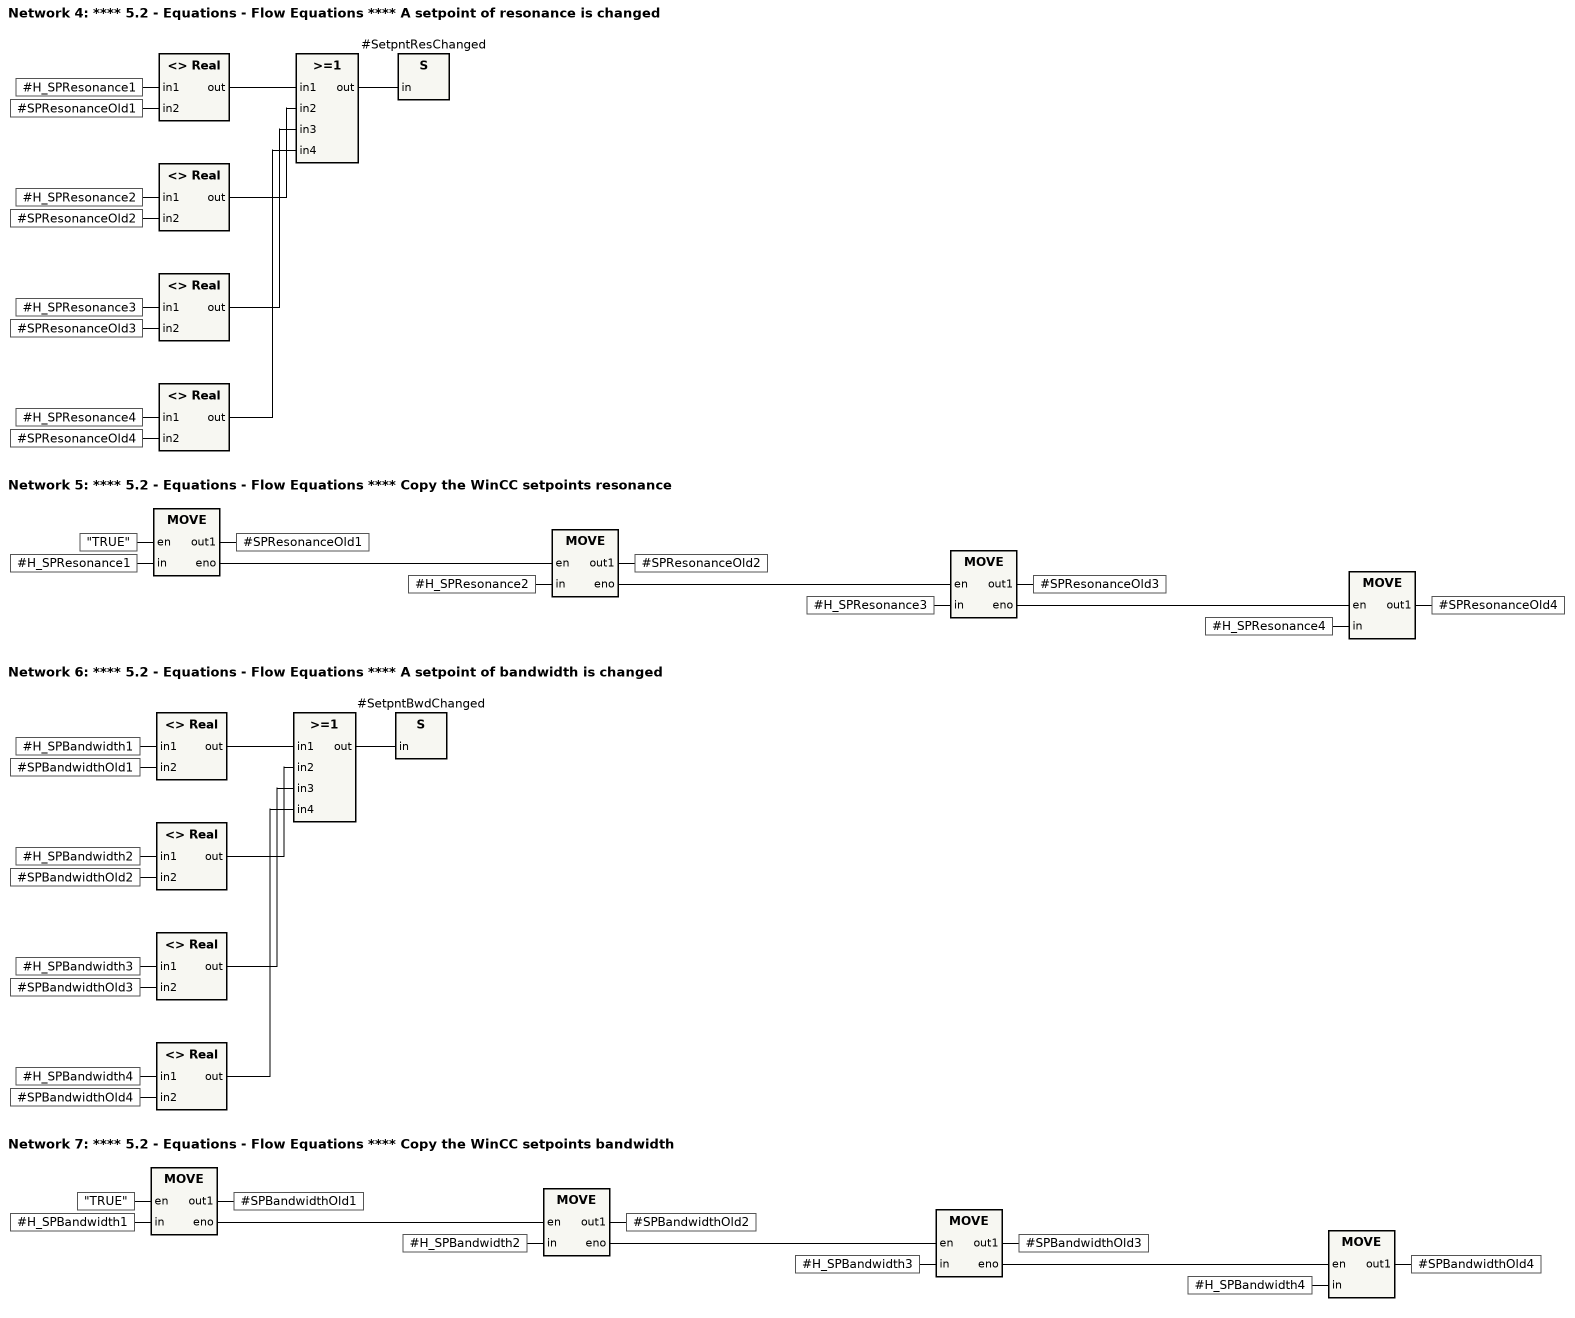
   IF (#H_SPResonance1 <> #SPResonanceOld1) OR (#H_SPResonance2 <> #SPResonanceOld2) OR (#H_SPResonance3 <> #SPResonanceOld3) OR (#H_SPResonance4 <> #SPResonanceOld4) THEN
       #SetpntResChanged := TRUE;
   END_IF;
END_REGION

REGION Network 5: **** 5.2 - Equations - Flow Equations **** Copy the WinCC setpoints resonance
   // Copy the WinCC setpoints resonance
   // ENO of a box is taken as its EN; it also drops when the box reports an error
   IF "TRUE" THEN
       #SPResonanceOld1 := #H_SPResonance1;
       #SPResonanceOld2 := #H_SPResonance2;
       #SPResonanceOld3 := #H_SPResonance3;
       #SPResonanceOld4 := #H_SPResonance4;
   END_IF;
END_REGION

REGION Network 6: **** 5.2 - Equations - Flow Equations **** A setpoint of bandwidth is changed
   // A setpoint of bandwidth is changed
   IF (#H_SPBandwidth1 <> #SPBandwidthOld1) OR (#H_SPBandwidth2 <> #SPBandwidthOld2) OR (#H_SPBandwidth3 <> #SPBandwidthOld3) OR (#H_SPBandwidth4 <> #SPBandwidthOld4) THEN
       #SetpntBwdChanged := TRUE;
   END_IF;
END_REGION

REGION Network 7: **** 5.2 - Equations - Flow Equations **** Copy the WinCC setpoints bandwidth
   // Copy the WinCC setpoints bandwidth
   // ENO of a box is taken as its EN; it also drops when the box reports an error
   IF "TRUE" THEN
       #SPBandwidthOld1 := #H_SPBandwidth1;
       #SPBandwidthOld2 := #H_SPBandwidth2;
       #SPBandwidthOld3 := #H_SPBandwidth3;
       #SPBandwidthOld4 := #H_SPBandwidth4;
   END_IF;
END_REGION

REGION Network 8: **** 5.2 - Equations - Flow Equations **** Selection Set-point 1
   // Selection Set-point 1
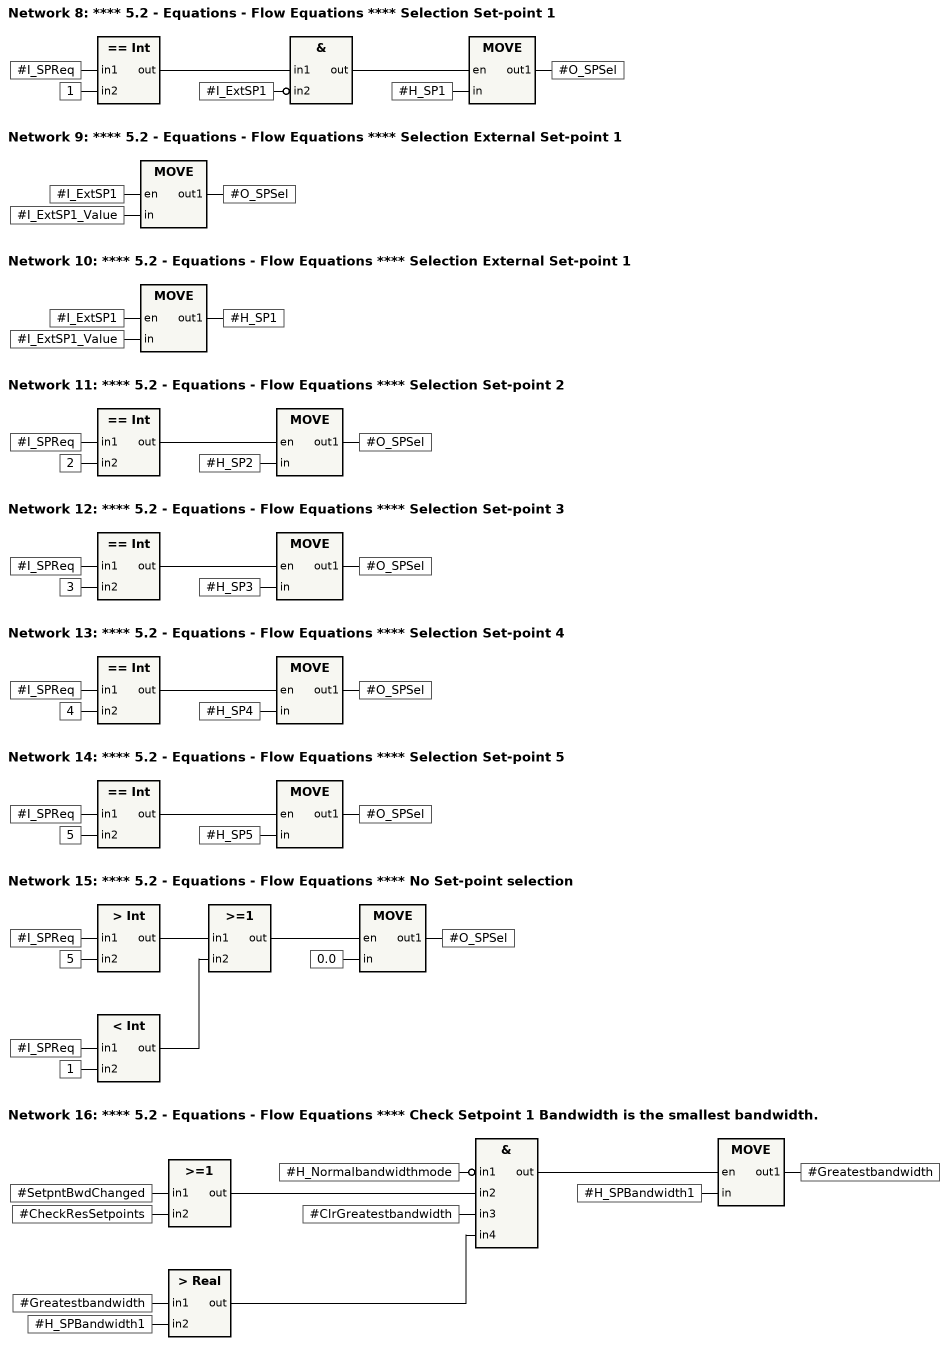
   IF (#I_SPReq = 1) AND NOT #I_ExtSP1 THEN #O_SPSel := #H_SP1; END_IF;
END_REGION

REGION Network 9: **** 5.2 - Equations - Flow Equations **** Selection External Set-point 1
   // Selection External Set-point 1
   IF #I_ExtSP1 THEN #O_SPSel := #I_ExtSP1_Value; END_IF;
END_REGION

REGION Network 10: **** 5.2 - Equations - Flow Equations **** Selection External Set-point 1
   // Selection External Set-point 1
   IF #I_ExtSP1 THEN #H_SP1 := #I_ExtSP1_Value; END_IF;
END_REGION

REGION Network 11: **** 5.2 - Equations - Flow Equations **** Selection Set-point 2
   // Selection Set-point 2
   IF #I_SPReq = 2 THEN #O_SPSel := #H_SP2; END_IF;
END_REGION

REGION Network 12: **** 5.2 - Equations - Flow Equations **** Selection Set-point 3
   // Selection Set-point 3
   IF #I_SPReq = 3 THEN #O_SPSel := #H_SP3; END_IF;
END_REGION

REGION Network 13: **** 5.2 - Equations - Flow Equations **** Selection Set-point 4
   // Selection Set-point 4
   IF #I_SPReq = 4 THEN #O_SPSel := #H_SP4; END_IF;
END_REGION

REGION Network 14: **** 5.2 - Equations - Flow Equations **** Selection Set-point 5
   // Selection Set-point 5
   IF #I_SPReq = 5 THEN #O_SPSel := #H_SP5; END_IF;
END_REGION

REGION Network 15: **** 5.2 - Equations - Flow Equations **** No Set-point selection
   // No Set-point selection
   IF (#I_SPReq > 5) OR (#I_SPReq < 1) THEN #O_SPSel := 0.0; END_IF;
END_REGION

REGION Network 16: **** 5.2 - Equations - Flow Equations **** Check Setpoint 1 Bandwidth is the smallest bandwidth.
   // Check Setpoint 1 Bandwidth is the smallest bandwidth.
   IF NOT #H_Normalbandwidthmode AND (#SetpntBwdChanged OR #CheckResSetpoints) AND #ClrGreatestbandwidth AND (#Greatestbandwidth > #H_SPBandwidth1) THEN
       #Greatestbandwidth := #H_SPBandwidth1;
   END_IF;
END_REGION

REGION Network 17: **** 5.2 - Equations - Flow Equations **** Check Setpoint 2 Bandwidth is the smallest bandwidth.
   // Check Setpoint 2 Bandwidth is the smallest bandwidth.
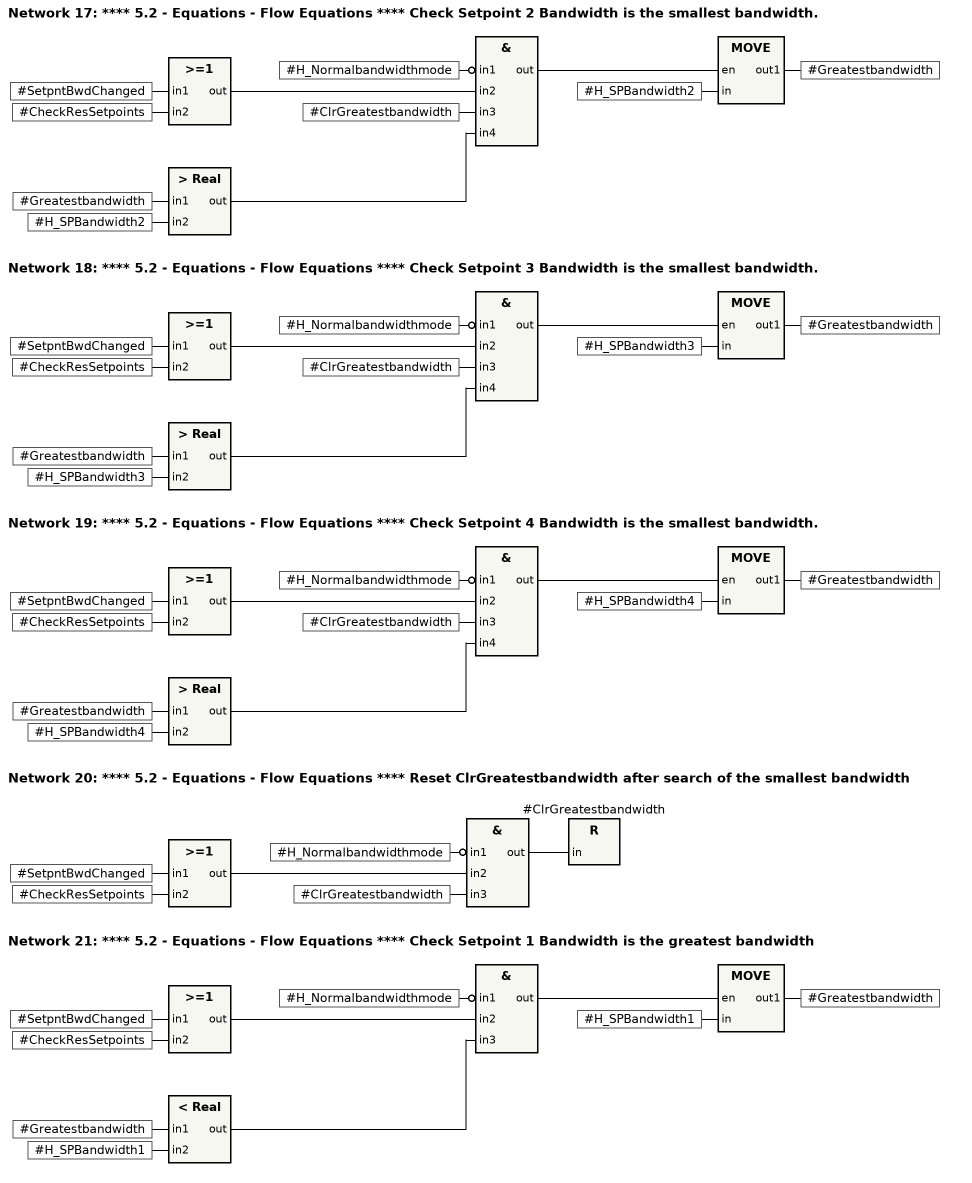
   IF NOT #H_Normalbandwidthmode AND (#SetpntBwdChanged OR #CheckResSetpoints) AND #ClrGreatestbandwidth AND (#Greatestbandwidth > #H_SPBandwidth2) THEN
       #Greatestbandwidth := #H_SPBandwidth2;
   END_IF;
END_REGION

REGION Network 18: **** 5.2 - Equations - Flow Equations **** Check Setpoint 3 Bandwidth is the smallest bandwidth.
   // Check Setpoint 3 Bandwidth is the smallest bandwidth.
   IF NOT #H_Normalbandwidthmode AND (#SetpntBwdChanged OR #CheckResSetpoints) AND #ClrGreatestbandwidth AND (#Greatestbandwidth > #H_SPBandwidth3) THEN
       #Greatestbandwidth := #H_SPBandwidth3;
   END_IF;
END_REGION

REGION Network 19: **** 5.2 - Equations - Flow Equations **** Check Setpoint 4 Bandwidth is the smallest bandwidth.
   // Check Setpoint 4 Bandwidth is the smallest bandwidth.
   IF NOT #H_Normalbandwidthmode AND (#SetpntBwdChanged OR #CheckResSetpoints) AND #ClrGreatestbandwidth AND (#Greatestbandwidth > #H_SPBandwidth4) THEN
       #Greatestbandwidth := #H_SPBandwidth4;
   END_IF;
END_REGION

REGION Network 20: **** 5.2 - Equations - Flow Equations **** Reset ClrGreatestbandwidth after search of the smallest bandwidth
   // Reset ClrGreatestbandwidth after search of the smallest bandwidth
   IF NOT #H_Normalbandwidthmode AND (#SetpntBwdChanged OR #CheckResSetpoints) AND #ClrGreatestbandwidth THEN
       #ClrGreatestbandwidth := FALSE;
   END_IF;
END_REGION

REGION Network 21: **** 5.2 - Equations - Flow Equations **** Check Setpoint 1 Bandwidth is the greatest bandwidth
   // Check Setpoint 1 Bandwidth is the greatest bandwidth
   IF NOT #H_Normalbandwidthmode AND (#SetpntBwdChanged OR #CheckResSetpoints) AND (#Greatestbandwidth < #H_SPBandwidth1) THEN
       #Greatestbandwidth := #H_SPBandwidth1;
   END_IF;
END_REGION

REGION Network 22: **** 5.2 - Equations - Flow Equations **** Check Setpoint 2 Bandwidth is the greatest bandwidth
   // Check Setpoint 2 Bandwidth is the greatest bandwidth
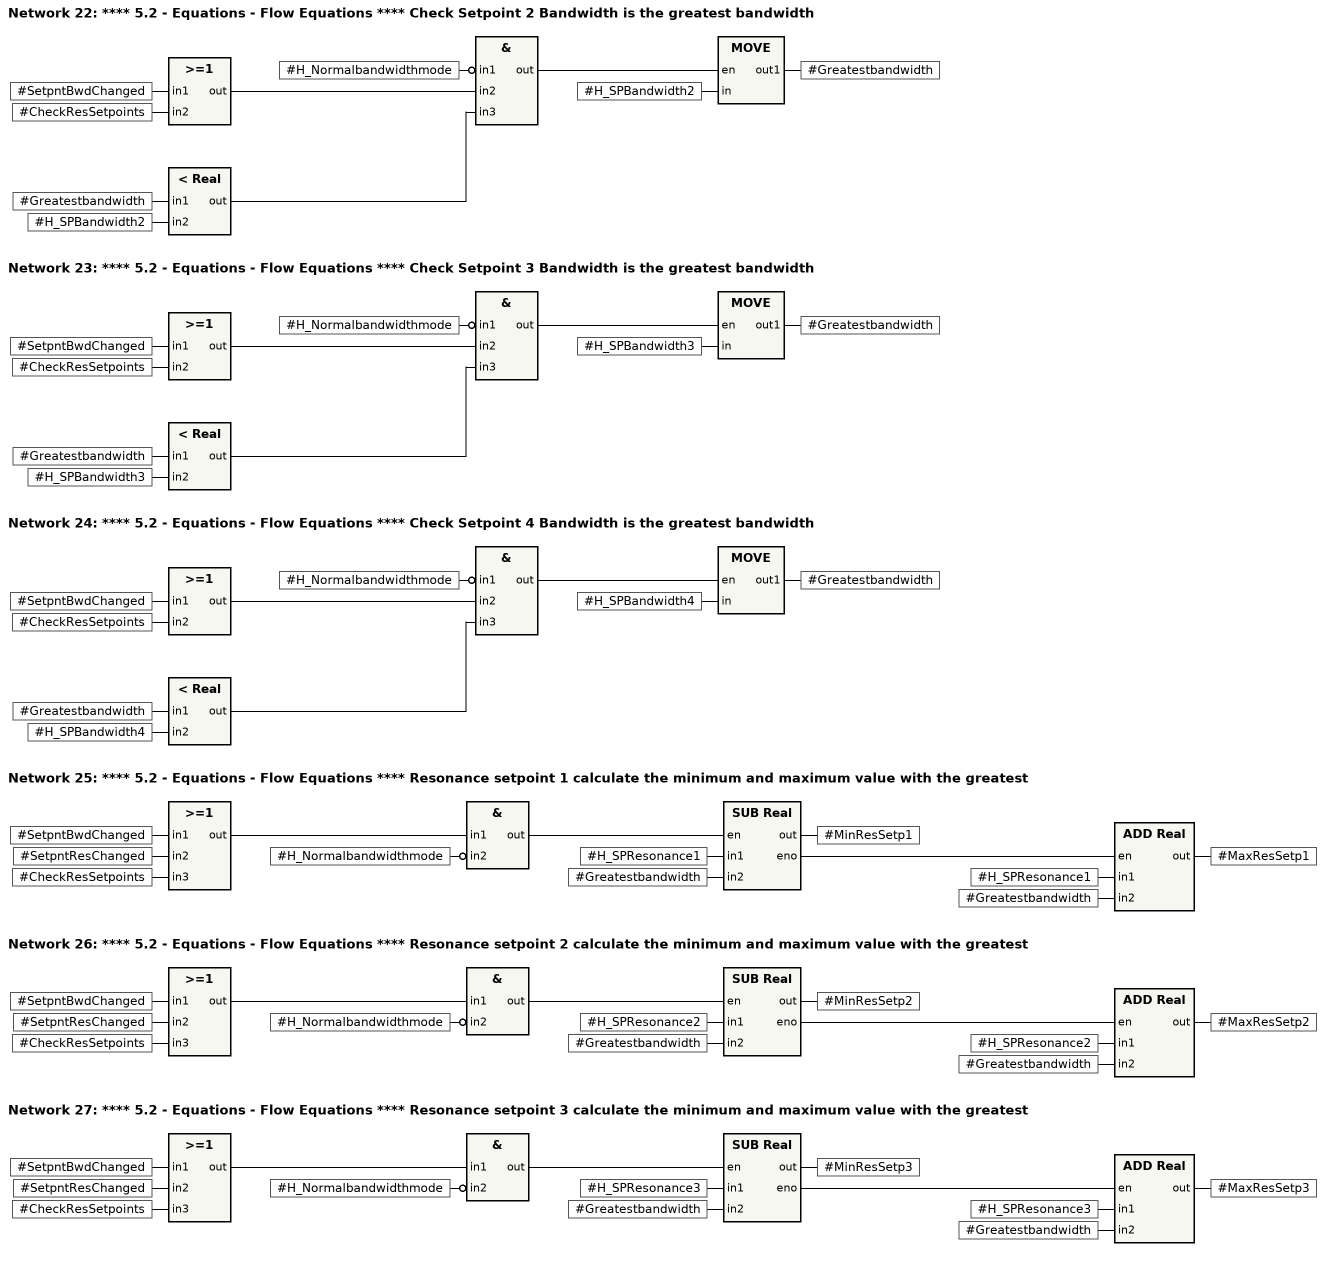
   IF NOT #H_Normalbandwidthmode AND (#SetpntBwdChanged OR #CheckResSetpoints) AND (#Greatestbandwidth < #H_SPBandwidth2) THEN
       #Greatestbandwidth := #H_SPBandwidth2;
   END_IF;
END_REGION

REGION Network 23: **** 5.2 - Equations - Flow Equations **** Check Setpoint 3 Bandwidth is the greatest bandwidth
   // Check Setpoint 3 Bandwidth is the greatest bandwidth
   IF NOT #H_Normalbandwidthmode AND (#SetpntBwdChanged OR #CheckResSetpoints) AND (#Greatestbandwidth < #H_SPBandwidth3) THEN
       #Greatestbandwidth := #H_SPBandwidth3;
   END_IF;
END_REGION

REGION Network 24: **** 5.2 - Equations - Flow Equations **** Check Setpoint 4 Bandwidth is the greatest bandwidth
   // Check Setpoint 4 Bandwidth is the greatest bandwidth
   IF NOT #H_Normalbandwidthmode AND (#SetpntBwdChanged OR #CheckResSetpoints) AND (#Greatestbandwidth < #H_SPBandwidth4) THEN
       #Greatestbandwidth := #H_SPBandwidth4;
   END_IF;
END_REGION

REGION Network 25: **** 5.2 - Equations - Flow Equations **** Resonance setpoint 1 calculate the minimum and maximum value with the greatest
   // Resonance setpoint 1 calculate the minimum and maximum value with the greatest 
   // bandwidth
   // ENO of a box is taken as its EN; it also drops when the box reports an error
   IF (#SetpntBwdChanged OR #SetpntResChanged OR #CheckResSetpoints) AND NOT #H_Normalbandwidthmode THEN
       #MinResSetp1 := #H_SPResonance1 - #Greatestbandwidth;
       #MaxResSetp1 := #H_SPResonance1 + #Greatestbandwidth;
   END_IF;
END_REGION

REGION Network 26: **** 5.2 - Equations - Flow Equations **** Resonance setpoint 2 calculate the minimum and maximum value with the greatest
   // Resonance setpoint 2 calculate the minimum and maximum value with the greatest 
   // bandwidth
   // ENO of a box is taken as its EN; it also drops when the box reports an error
   IF (#SetpntBwdChanged OR #SetpntResChanged OR #CheckResSetpoints) AND NOT #H_Normalbandwidthmode THEN
       #MinResSetp2 := #H_SPResonance2 - #Greatestbandwidth;
       #MaxResSetp2 := #H_SPResonance2 + #Greatestbandwidth;
   END_IF;
END_REGION

REGION Network 27: **** 5.2 - Equations - Flow Equations **** Resonance setpoint 3 calculate the minimum and maximum value with the greatest
   // Resonance setpoint 3 calculate the minimum and maximum value with the greatest 
   // bandwidth
   // ENO of a box is taken as its EN; it also drops when the box reports an error
   IF (#SetpntBwdChanged OR #SetpntResChanged OR #CheckResSetpoints) AND NOT #H_Normalbandwidthmode THEN
       #MinResSetp3 := #H_SPResonance3 - #Greatestbandwidth;
       #MaxResSetp3 := #H_SPResonance3 + #Greatestbandwidth;
   END_IF;
END_REGION

REGION Network 28: **** 5.2 - Equations - Flow Equations **** Resonance setpoint 4 calculate the minimum and maximum value with the greatest
   // Resonance setpoint 4 calculate the minimum and maximum value with the greatest 
   // bandwidth
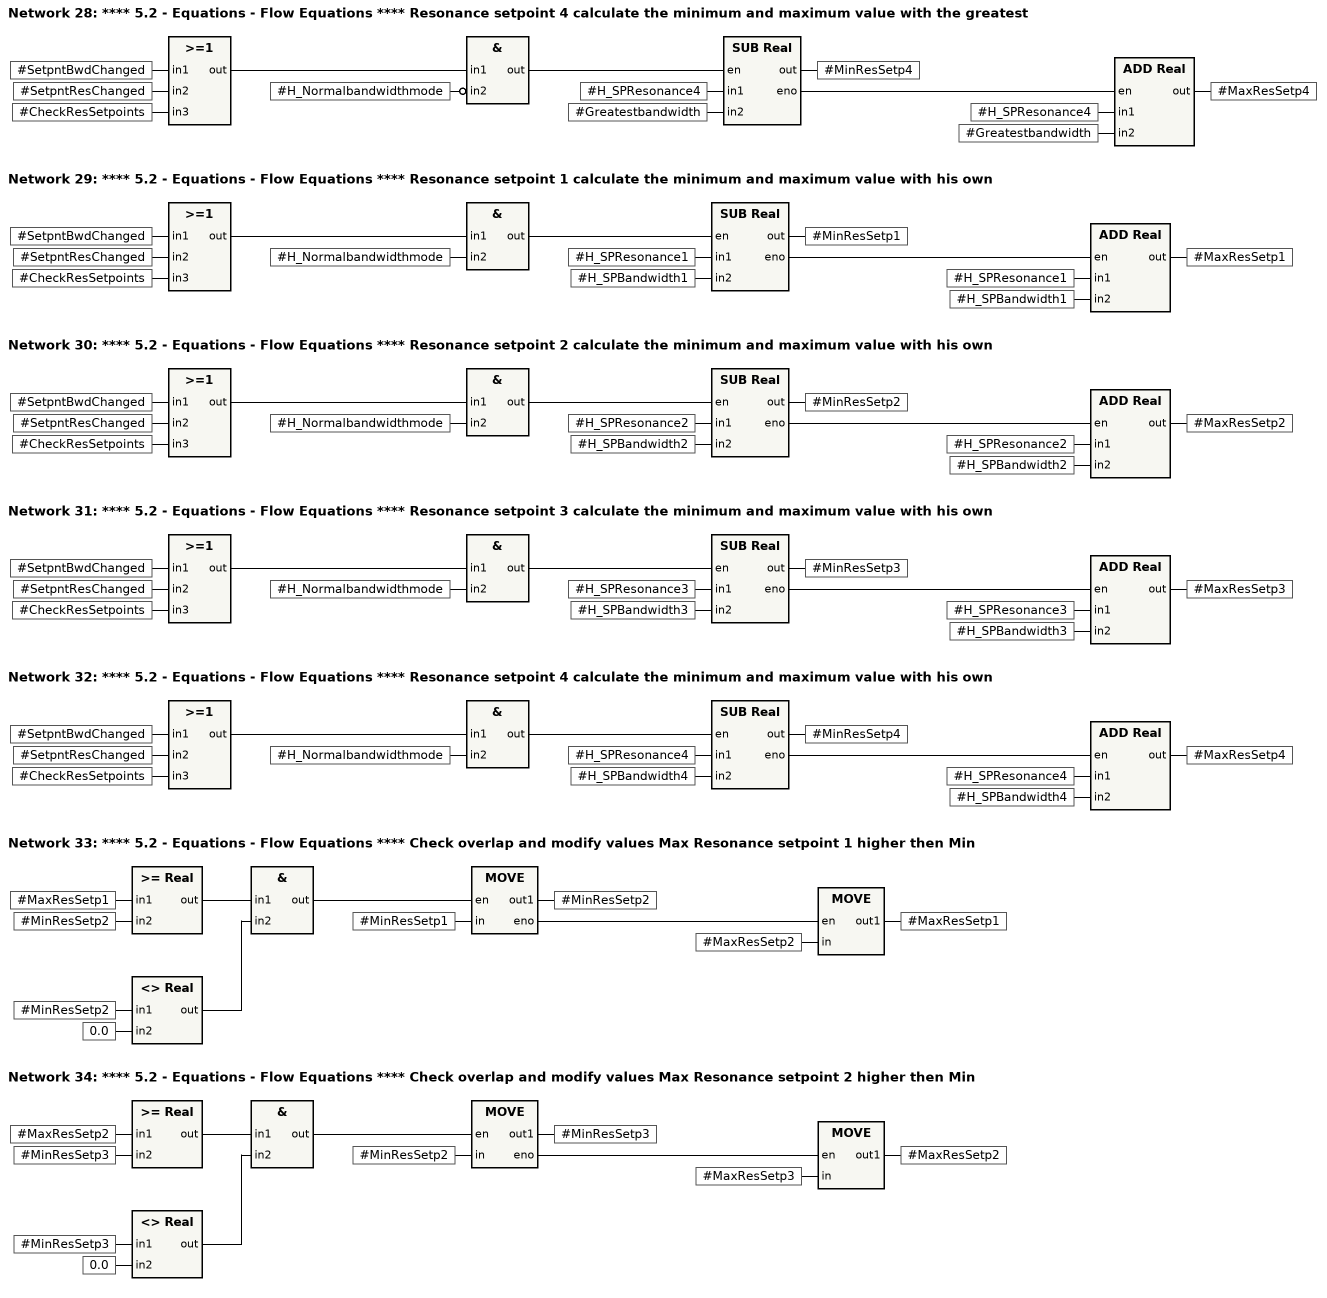
   // ENO of a box is taken as its EN; it also drops when the box reports an error
   IF (#SetpntBwdChanged OR #SetpntResChanged OR #CheckResSetpoints) AND NOT #H_Normalbandwidthmode THEN
       #MinResSetp4 := #H_SPResonance4 - #Greatestbandwidth;
       #MaxResSetp4 := #H_SPResonance4 + #Greatestbandwidth;
   END_IF;
END_REGION

REGION Network 29: **** 5.2 - Equations - Flow Equations **** Resonance setpoint 1 calculate the minimum and maximum value with his own
   // Resonance setpoint 1 calculate the minimum and maximum value with his own 
   // bandwidth
   // ENO of a box is taken as its EN; it also drops when the box reports an error
   IF (#SetpntBwdChanged OR #SetpntResChanged OR #CheckResSetpoints) AND #H_Normalbandwidthmode THEN
       #MinResSetp1 := #H_SPResonance1 - #H_SPBandwidth1;
       #MaxResSetp1 := #H_SPResonance1 + #H_SPBandwidth1;
   END_IF;
END_REGION

REGION Network 30: **** 5.2 - Equations - Flow Equations **** Resonance setpoint 2 calculate the minimum and maximum value with his own
   // Resonance setpoint 2 calculate the minimum and maximum value with his own 
   // bandwidth
   // ENO of a box is taken as its EN; it also drops when the box reports an error
   IF (#SetpntBwdChanged OR #SetpntResChanged OR #CheckResSetpoints) AND #H_Normalbandwidthmode THEN
       #MinResSetp2 := #H_SPResonance2 - #H_SPBandwidth2;
       #MaxResSetp2 := #H_SPResonance2 + #H_SPBandwidth2;
   END_IF;
END_REGION

REGION Network 31: **** 5.2 - Equations - Flow Equations **** Resonance setpoint 3 calculate the minimum and maximum value with his own
   // Resonance setpoint 3 calculate the minimum and maximum value with his own 
   // bandwidth
   // ENO of a box is taken as its EN; it also drops when the box reports an error
   IF (#SetpntBwdChanged OR #SetpntResChanged OR #CheckResSetpoints) AND #H_Normalbandwidthmode THEN
       #MinResSetp3 := #H_SPResonance3 - #H_SPBandwidth3;
       #MaxResSetp3 := #H_SPResonance3 + #H_SPBandwidth3;
   END_IF;
END_REGION

REGION Network 32: **** 5.2 - Equations - Flow Equations **** Resonance setpoint 4 calculate the minimum and maximum value with his own
   // Resonance setpoint 4 calculate the minimum and maximum value with his own 
   // bandwidth
   // ENO of a box is taken as its EN; it also drops when the box reports an error
   IF (#SetpntBwdChanged OR #SetpntResChanged OR #CheckResSetpoints) AND #H_Normalbandwidthmode THEN
       #MinResSetp4 := #H_SPResonance4 - #H_SPBandwidth4;
       #MaxResSetp4 := #H_SPResonance4 + #H_SPBandwidth4;
   END_IF;
END_REGION

REGION Network 33: **** 5.2 - Equations - Flow Equations **** Check overlap and modify values Max Resonance setpoint 1 higher then Min
   // Check overlap and modify values Max Resonance setpoint 1 higher then Min 
   // Resonance setpoint 2
   // ENO of a box is taken as its EN; it also drops when the box reports an error
   #_w1 := (#MaxResSetp1 >= #MinResSetp2) AND (#MinResSetp2 <> 0.0);
   IF #_w1 THEN
       #MinResSetp2 := #MinResSetp1;
       #MaxResSetp1 := #MaxResSetp2;
   END_IF;
END_REGION

REGION Network 34: **** 5.2 - Equations - Flow Equations **** Check overlap and modify values Max Resonance setpoint 2 higher then Min
   // Check overlap and modify values Max Resonance setpoint 2 higher then Min 
   // Resonance setpoint 3
   // ENO of a box is taken as its EN; it also drops when the box reports an error
   #_w1 := (#MaxResSetp2 >= #MinResSetp3) AND (#MinResSetp3 <> 0.0);
   IF #_w1 THEN
       #MinResSetp3 := #MinResSetp2;
       #MaxResSetp2 := #MaxResSetp3;
   END_IF;
END_REGION

REGION Network 35: **** 5.2 - Equations - Flow Equations **** Check overlap and modify values Max Resonance setpoint 3 higher then Min
   // Check overlap and modify values Max Resonance setpoint 3 higher then Min 
   // Resonance setpoint 4
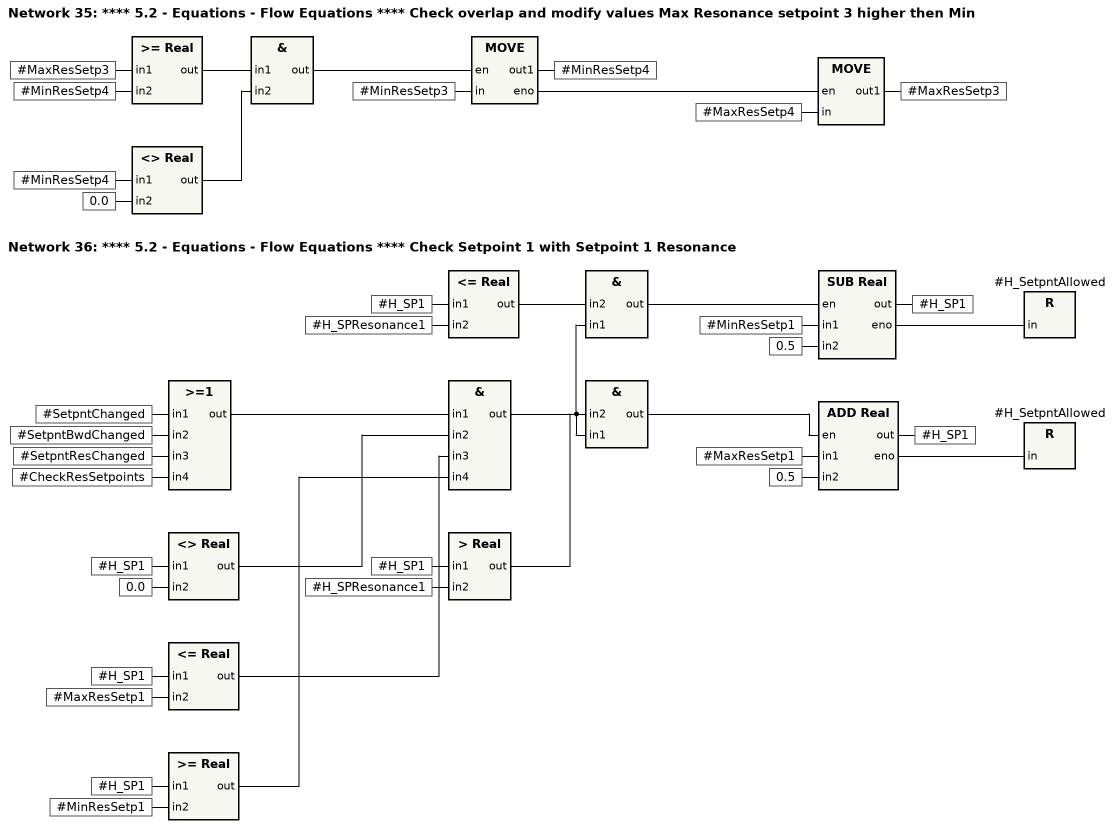
   // ENO of a box is taken as its EN; it also drops when the box reports an error
   #_w1 := (#MaxResSetp3 >= #MinResSetp4) AND (#MinResSetp4 <> 0.0);
   IF #_w1 THEN
       #MinResSetp4 := #MinResSetp3;
       #MaxResSetp3 := #MaxResSetp4;
   END_IF;
END_REGION

REGION Network 36: **** 5.2 - Equations - Flow Equations **** Check Setpoint 1 with Setpoint 1 Resonance
   // Check Setpoint 1 with Setpoint 1 Resonance 
   // Setpoint 1 is no longer allowed, calculate prefered allowed setpoint 1
   // ENO of a box is taken as its EN; it also drops when the box reports an error
   #_w1 := (#SetpntChanged OR #SetpntBwdChanged OR #SetpntResChanged OR #CheckResSetpoints) AND (#H_SP1 <> 0.0) AND (#H_SP1 <= #MaxResSetp1) AND (#H_SP1 >= #MinResSetp1);
   #_w2 := (#H_SP1 <= #H_SPResonance1) AND #_w1;
   IF #_w2 THEN
       #H_SP1 := #MinResSetp1 - 0.5;
       #H_SetpntAllowed := FALSE;
   END_IF;
   #_w3 := (#H_SP1 > #H_SPResonance1) AND #_w1;
   IF #_w3 THEN
       #H_SP1 := #MaxResSetp1 + 0.5;
       #H_SetpntAllowed := FALSE;
   END_IF;
END_REGION

REGION Network 37: **** 5.2 - Equations - Flow Equations **** Check Setpoint 1 with Setpoint 2 Resonance
   // Check Setpoint 1 with Setpoint 2 Resonance 
   // Setpoint 1 is no longer allowed, calculate prefered allowed setpoint 1
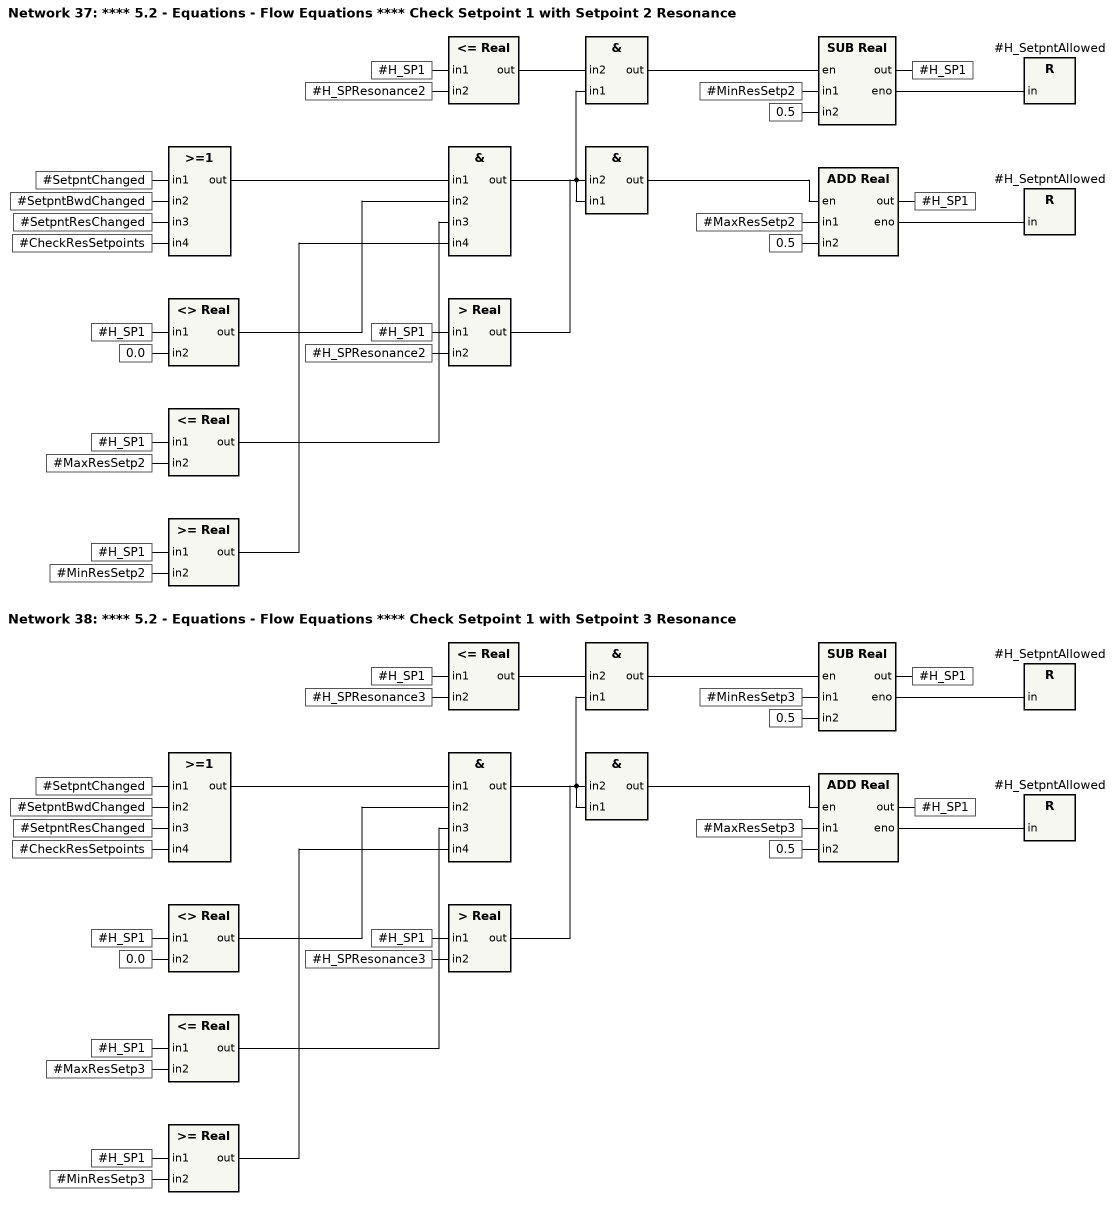
   // ENO of a box is taken as its EN; it also drops when the box reports an error
   #_w1 := (#SetpntChanged OR #SetpntBwdChanged OR #SetpntResChanged OR #CheckResSetpoints) AND (#H_SP1 <> 0.0) AND (#H_SP1 <= #MaxResSetp2) AND (#H_SP1 >= #MinResSetp2);
   #_w2 := (#H_SP1 <= #H_SPResonance2) AND #_w1;
   IF #_w2 THEN
       #H_SP1 := #MinResSetp2 - 0.5;
       #H_SetpntAllowed := FALSE;
   END_IF;
   #_w3 := (#H_SP1 > #H_SPResonance2) AND #_w1;
   IF #_w3 THEN
       #H_SP1 := #MaxResSetp2 + 0.5;
       #H_SetpntAllowed := FALSE;
   END_IF;
END_REGION

REGION Network 38: **** 5.2 - Equations - Flow Equations **** Check Setpoint 1 with Setpoint 3 Resonance
   // Check Setpoint 1 with Setpoint 3 Resonance 
   // Setpoint 1 is no longer allowed, calculate prefered allowed setpoint 1
   // ENO of a box is taken as its EN; it also drops when the box reports an error
   #_w1 := (#SetpntChanged OR #SetpntBwdChanged OR #SetpntResChanged OR #CheckResSetpoints) AND (#H_SP1 <> 0.0) AND (#H_SP1 <= #MaxResSetp3) AND (#H_SP1 >= #MinResSetp3);
   #_w2 := (#H_SP1 <= #H_SPResonance3) AND #_w1;
   IF #_w2 THEN
       #H_SP1 := #MinResSetp3 - 0.5;
       #H_SetpntAllowed := FALSE;
   END_IF;
   #_w3 := (#H_SP1 > #H_SPResonance3) AND #_w1;
   IF #_w3 THEN
       #H_SP1 := #MaxResSetp3 + 0.5;
       #H_SetpntAllowed := FALSE;
   END_IF;
END_REGION

REGION Network 39: **** 5.2 - Equations - Flow Equations **** Check Setpoint 1 with Setpoint 4 Resonance
   // Check Setpoint 1 with Setpoint 4 Resonance 
   // Setpoint 1 is no longer allowed, calculate prefered allowed setpoint 1
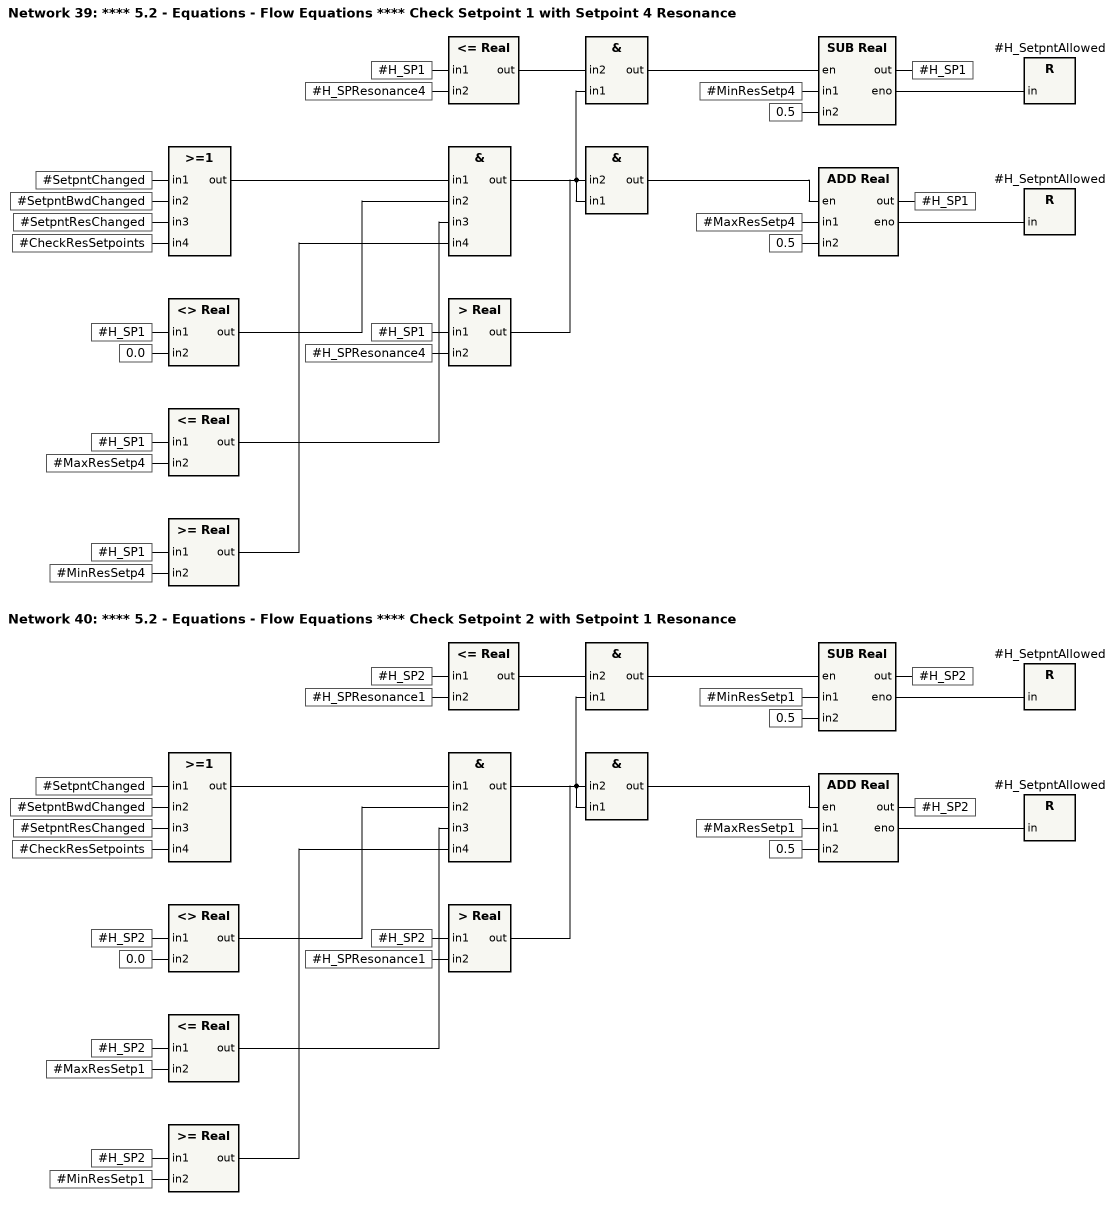
   // ENO of a box is taken as its EN; it also drops when the box reports an error
   #_w1 := (#SetpntChanged OR #SetpntBwdChanged OR #SetpntResChanged OR #CheckResSetpoints) AND (#H_SP1 <> 0.0) AND (#H_SP1 <= #MaxResSetp4) AND (#H_SP1 >= #MinResSetp4);
   #_w2 := (#H_SP1 <= #H_SPResonance4) AND #_w1;
   IF #_w2 THEN
       #H_SP1 := #MinResSetp4 - 0.5;
       #H_SetpntAllowed := FALSE;
   END_IF;
   #_w3 := (#H_SP1 > #H_SPResonance4) AND #_w1;
   IF #_w3 THEN
       #H_SP1 := #MaxResSetp4 + 0.5;
       #H_SetpntAllowed := FALSE;
   END_IF;
END_REGION

REGION Network 40: **** 5.2 - Equations - Flow Equations **** Check Setpoint 2 with Setpoint 1 Resonance
   // Check Setpoint 2 with Setpoint 1 Resonance 
   // Setpoint 2 is no longer allowed, calculate prefered allowed setpoint 2
   // ENO of a box is taken as its EN; it also drops when the box reports an error
   #_w1 := (#SetpntChanged OR #SetpntBwdChanged OR #SetpntResChanged OR #CheckResSetpoints) AND (#H_SP2 <> 0.0) AND (#H_SP2 <= #MaxResSetp1) AND (#H_SP2 >= #MinResSetp1);
   #_w2 := (#H_SP2 <= #H_SPResonance1) AND #_w1;
   IF #_w2 THEN
       #H_SP2 := #MinResSetp1 - 0.5;
       #H_SetpntAllowed := FALSE;
   END_IF;
   #_w3 := (#H_SP2 > #H_SPResonance1) AND #_w1;
   IF #_w3 THEN
       #H_SP2 := #MaxResSetp1 + 0.5;
       #H_SetpntAllowed := FALSE;
   END_IF;
END_REGION

REGION Network 41: **** 5.2 - Equations - Flow Equations **** Check Setpoint 2 with Setpoint 2 Resonance
   // Check Setpoint 2 with Setpoint 2 Resonance 
   // Setpoint 2 is no longer allowed, calculate prefered allowed setpoint 2
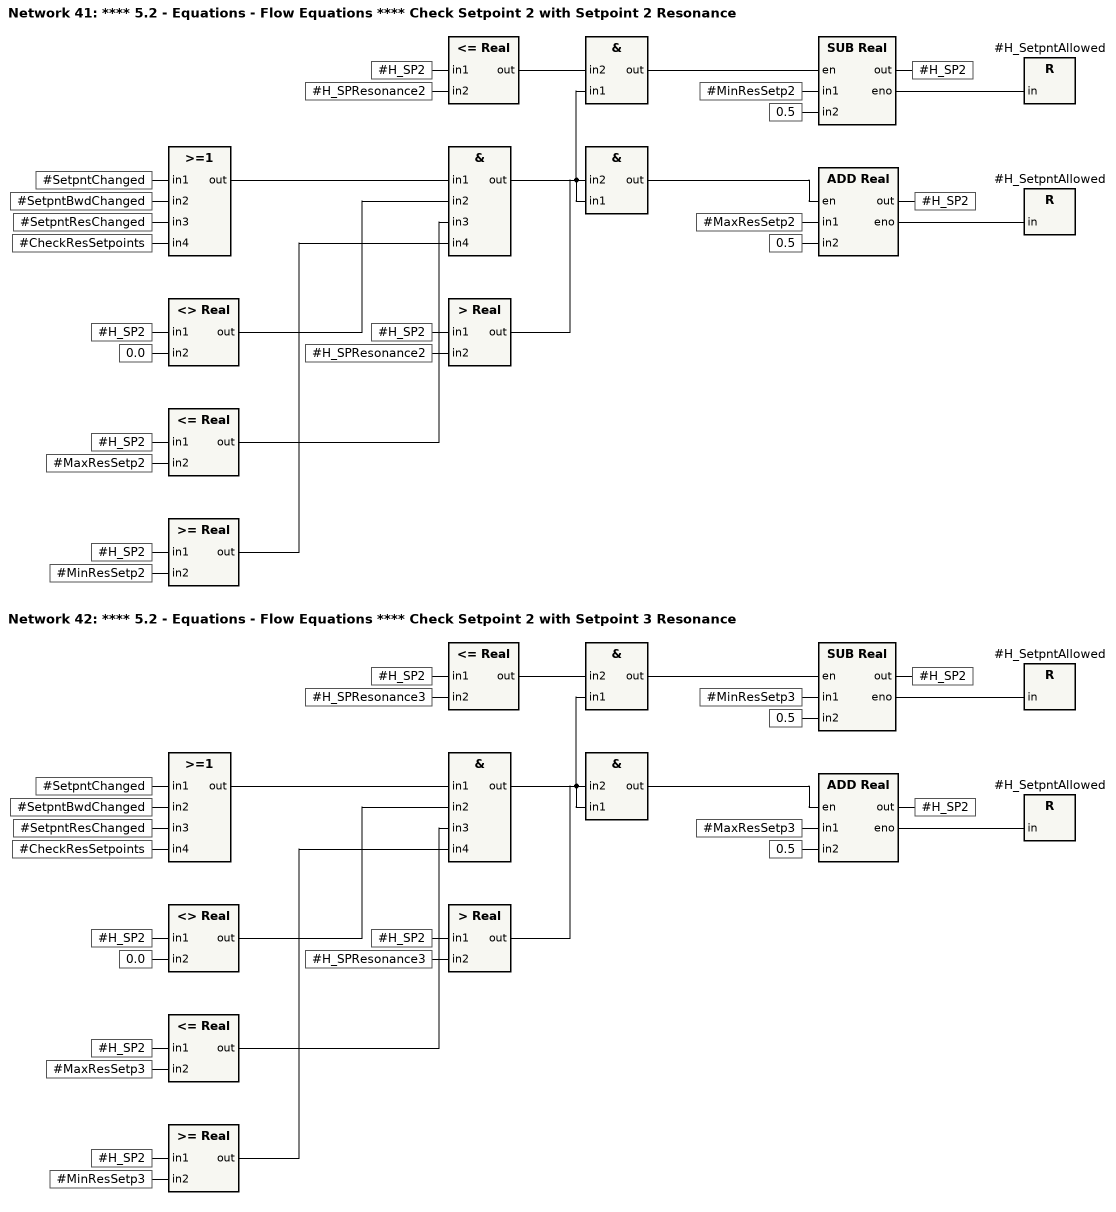
   // ENO of a box is taken as its EN; it also drops when the box reports an error
   #_w1 := (#SetpntChanged OR #SetpntBwdChanged OR #SetpntResChanged OR #CheckResSetpoints) AND (#H_SP2 <> 0.0) AND (#H_SP2 <= #MaxResSetp2) AND (#H_SP2 >= #MinResSetp2);
   #_w2 := (#H_SP2 <= #H_SPResonance2) AND #_w1;
   IF #_w2 THEN
       #H_SP2 := #MinResSetp2 - 0.5;
       #H_SetpntAllowed := FALSE;
   END_IF;
   #_w3 := (#H_SP2 > #H_SPResonance2) AND #_w1;
   IF #_w3 THEN
       #H_SP2 := #MaxResSetp2 + 0.5;
       #H_SetpntAllowed := FALSE;
   END_IF;
END_REGION

REGION Network 42: **** 5.2 - Equations - Flow Equations **** Check Setpoint 2 with Setpoint 3 Resonance
   // Check Setpoint 2 with Setpoint 3 Resonance 
   // Setpoint 2 is no longer allowed, calculate prefered allowed setpoint 2
   // ENO of a box is taken as its EN; it also drops when the box reports an error
   #_w1 := (#SetpntChanged OR #SetpntBwdChanged OR #SetpntResChanged OR #CheckResSetpoints) AND (#H_SP2 <> 0.0) AND (#H_SP2 <= #MaxResSetp3) AND (#H_SP2 >= #MinResSetp3);
   #_w2 := (#H_SP2 <= #H_SPResonance3) AND #_w1;
   IF #_w2 THEN
       #H_SP2 := #MinResSetp3 - 0.5;
       #H_SetpntAllowed := FALSE;
   END_IF;
   #_w3 := (#H_SP2 > #H_SPResonance3) AND #_w1;
   IF #_w3 THEN
       #H_SP2 := #MaxResSetp3 + 0.5;
       #H_SetpntAllowed := FALSE;
   END_IF;
END_REGION

REGION Network 43: **** 5.2 - Equations - Flow Equations **** Check Setpoint 2 with Setpoint 4 Resonance
   // Check Setpoint 2 with Setpoint 4 Resonance 
   // Setpoint 2 is no longer allowed, calculate prefered allowed setpoint 2
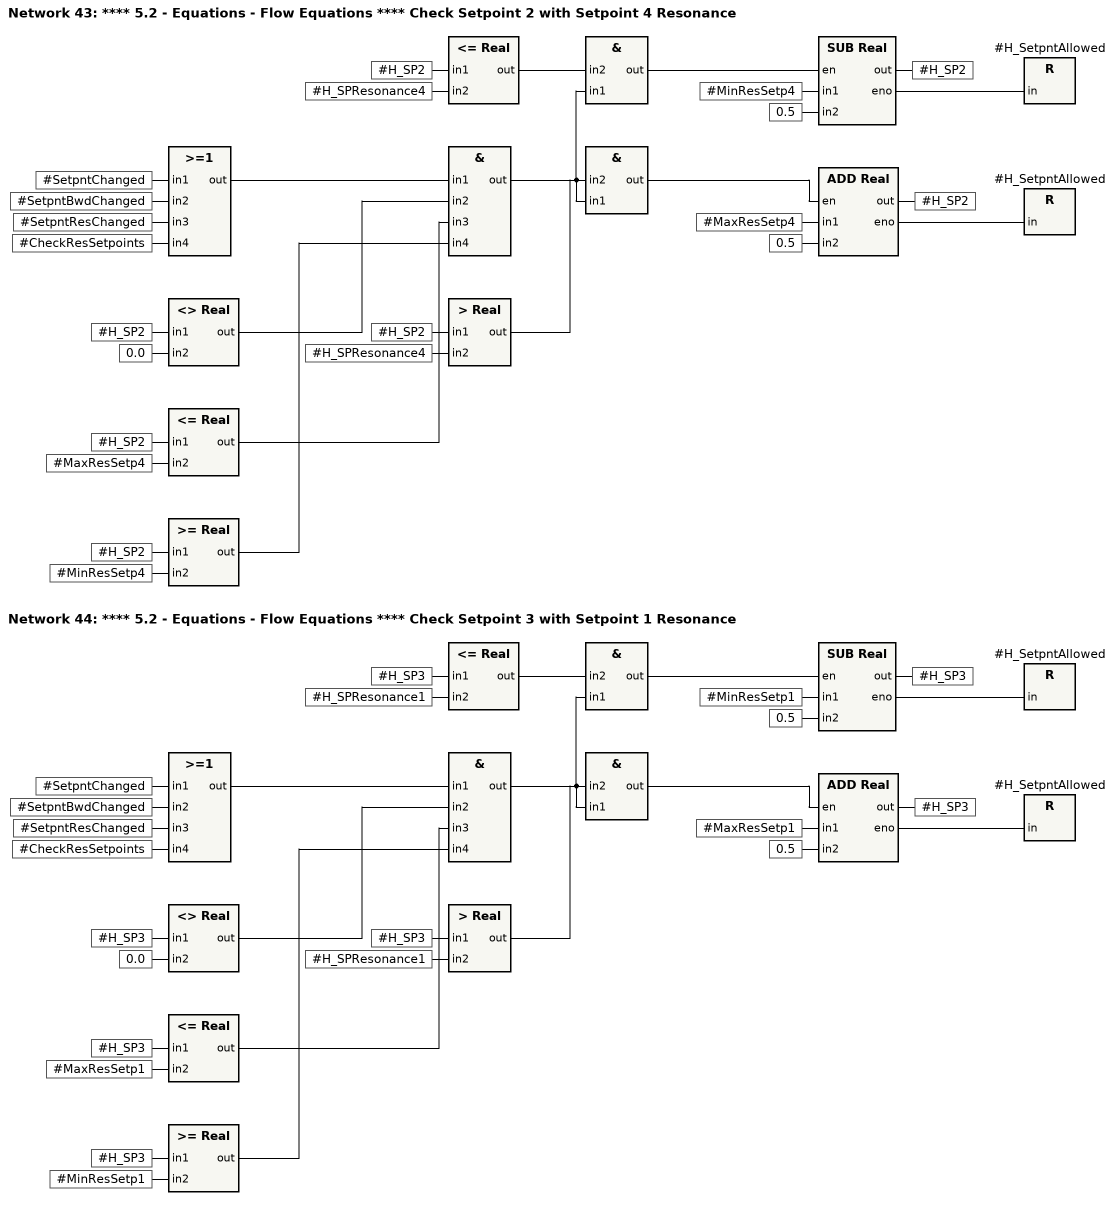
   // ENO of a box is taken as its EN; it also drops when the box reports an error
   #_w1 := (#SetpntChanged OR #SetpntBwdChanged OR #SetpntResChanged OR #CheckResSetpoints) AND (#H_SP2 <> 0.0) AND (#H_SP2 <= #MaxResSetp4) AND (#H_SP2 >= #MinResSetp4);
   #_w2 := (#H_SP2 <= #H_SPResonance4) AND #_w1;
   IF #_w2 THEN
       #H_SP2 := #MinResSetp4 - 0.5;
       #H_SetpntAllowed := FALSE;
   END_IF;
   #_w3 := (#H_SP2 > #H_SPResonance4) AND #_w1;
   IF #_w3 THEN
       #H_SP2 := #MaxResSetp4 + 0.5;
       #H_SetpntAllowed := FALSE;
   END_IF;
END_REGION

REGION Network 44: **** 5.2 - Equations - Flow Equations **** Check Setpoint 3 with Setpoint 1 Resonance
   // Check Setpoint 3 with Setpoint 1 Resonance 
   // Setpoint 3 is no longer allowed, calculate prefered allowed setpoint 3
   // ENO of a box is taken as its EN; it also drops when the box reports an error
   #_w1 := (#SetpntChanged OR #SetpntBwdChanged OR #SetpntResChanged OR #CheckResSetpoints) AND (#H_SP3 <> 0.0) AND (#H_SP3 <= #MaxResSetp1) AND (#H_SP3 >= #MinResSetp1);
   #_w2 := (#H_SP3 <= #H_SPResonance1) AND #_w1;
   IF #_w2 THEN
       #H_SP3 := #MinResSetp1 - 0.5;
       #H_SetpntAllowed := FALSE;
   END_IF;
   #_w3 := (#H_SP3 > #H_SPResonance1) AND #_w1;
   IF #_w3 THEN
       #H_SP3 := #MaxResSetp1 + 0.5;
       #H_SetpntAllowed := FALSE;
   END_IF;
END_REGION

REGION Network 45: **** 5.2 - Equations - Flow Equations **** Check Setpoint 3 with Setpoint 2 Resonance
   // Check Setpoint 3 with Setpoint 2 Resonance 
   // Setpoint 3 is no longer allowed, calculate prefered allowed setpoint 3
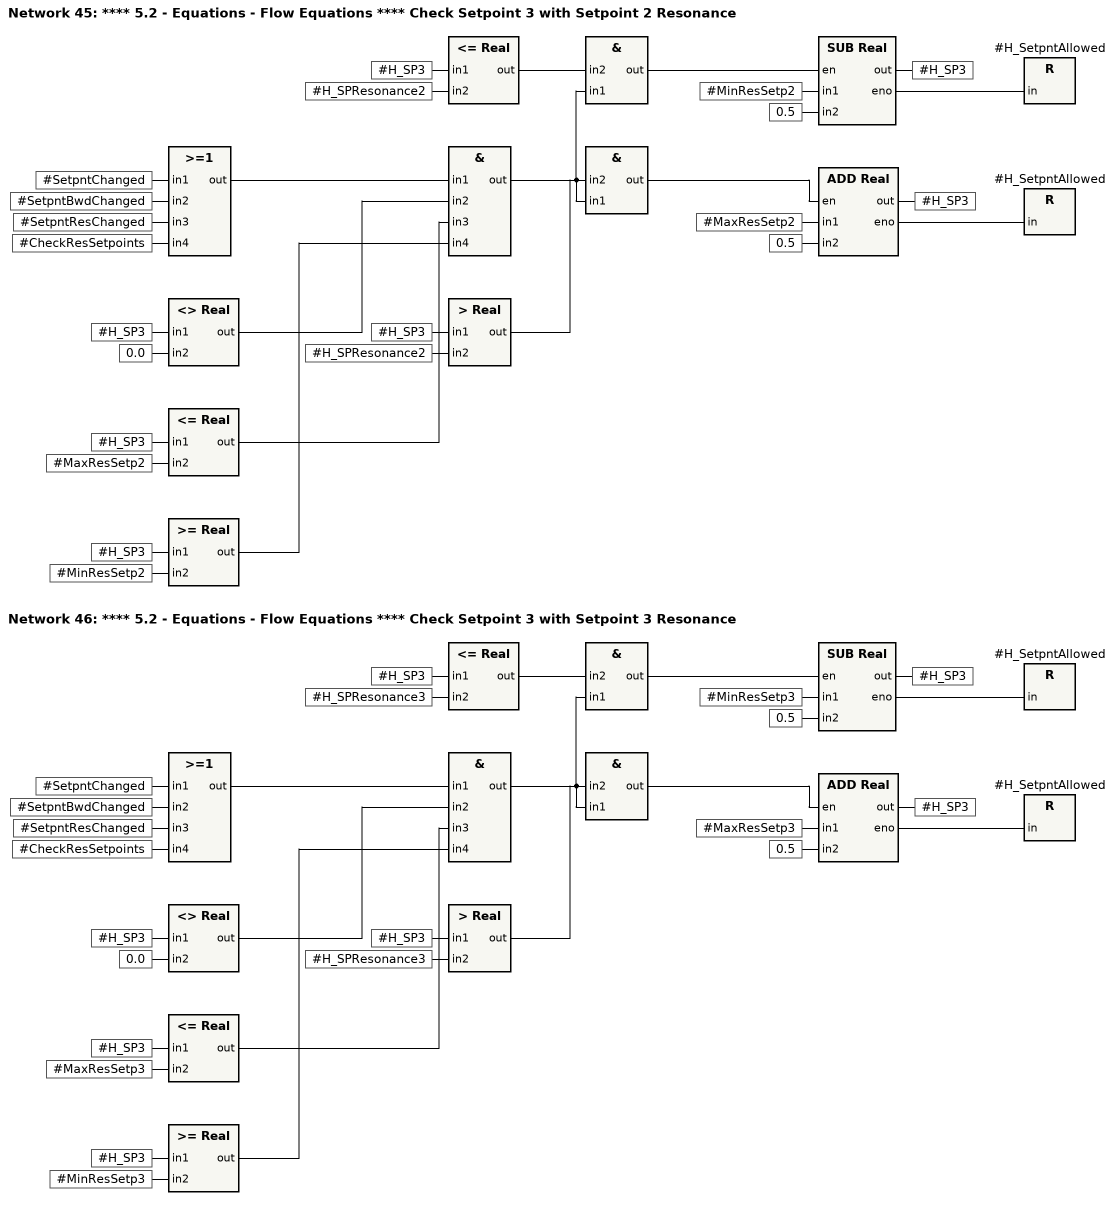
   // ENO of a box is taken as its EN; it also drops when the box reports an error
   #_w1 := (#SetpntChanged OR #SetpntBwdChanged OR #SetpntResChanged OR #CheckResSetpoints) AND (#H_SP3 <> 0.0) AND (#H_SP3 <= #MaxResSetp2) AND (#H_SP3 >= #MinResSetp2);
   #_w2 := (#H_SP3 <= #H_SPResonance2) AND #_w1;
   IF #_w2 THEN
       #H_SP3 := #MinResSetp2 - 0.5;
       #H_SetpntAllowed := FALSE;
   END_IF;
   #_w3 := (#H_SP3 > #H_SPResonance2) AND #_w1;
   IF #_w3 THEN
       #H_SP3 := #MaxResSetp2 + 0.5;
       #H_SetpntAllowed := FALSE;
   END_IF;
END_REGION

REGION Network 46: **** 5.2 - Equations - Flow Equations **** Check Setpoint 3 with Setpoint 3 Resonance
   // Check Setpoint 3 with Setpoint 3 Resonance 
   // Setpoint 3 is no longer allowed, calculate prefered allowed setpoint 3
   // ENO of a box is taken as its EN; it also drops when the box reports an error
   #_w1 := (#SetpntChanged OR #SetpntBwdChanged OR #SetpntResChanged OR #CheckResSetpoints) AND (#H_SP3 <> 0.0) AND (#H_SP3 <= #MaxResSetp3) AND (#H_SP3 >= #MinResSetp3);
   #_w2 := (#H_SP3 <= #H_SPResonance3) AND #_w1;
   IF #_w2 THEN
       #H_SP3 := #MinResSetp3 - 0.5;
       #H_SetpntAllowed := FALSE;
   END_IF;
   #_w3 := (#H_SP3 > #H_SPResonance3) AND #_w1;
   IF #_w3 THEN
       #H_SP3 := #MaxResSetp3 + 0.5;
       #H_SetpntAllowed := FALSE;
   END_IF;
END_REGION

REGION Network 47: **** 5.2 - Equations - Flow Equations **** Check Setpoint 3 with Setpoint 4 Resonance
   // Check Setpoint 3 with Setpoint 4 Resonance 
   // Setpoint 3 is no longer allowed, calculate prefered allowed setpoint 3
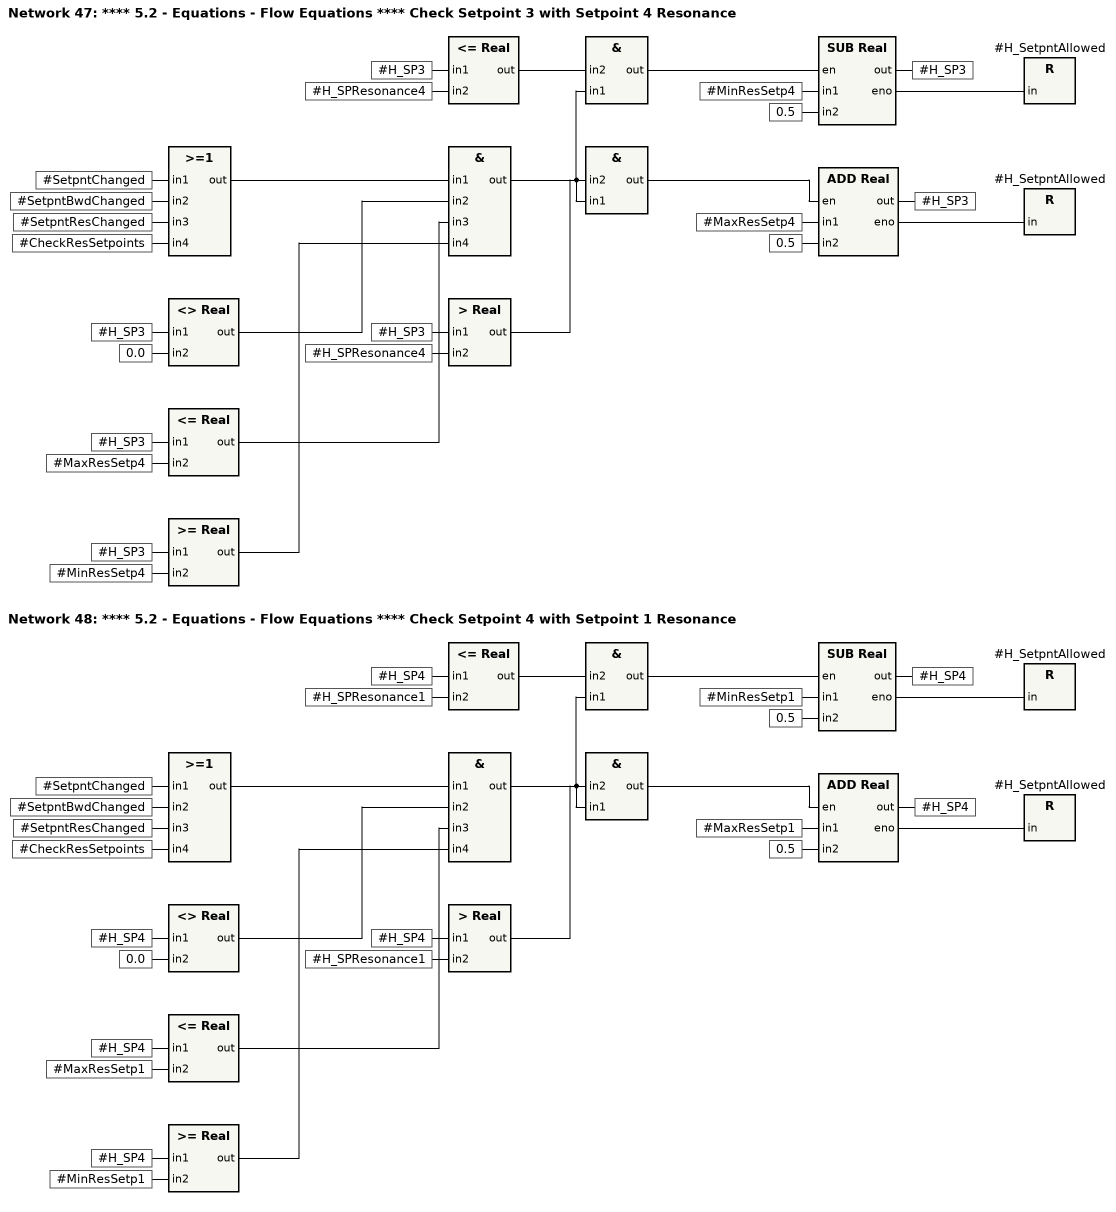
   // ENO of a box is taken as its EN; it also drops when the box reports an error
   #_w1 := (#SetpntChanged OR #SetpntBwdChanged OR #SetpntResChanged OR #CheckResSetpoints) AND (#H_SP3 <> 0.0) AND (#H_SP3 <= #MaxResSetp4) AND (#H_SP3 >= #MinResSetp4);
   #_w2 := (#H_SP3 <= #H_SPResonance4) AND #_w1;
   IF #_w2 THEN
       #H_SP3 := #MinResSetp4 - 0.5;
       #H_SetpntAllowed := FALSE;
   END_IF;
   #_w3 := (#H_SP3 > #H_SPResonance4) AND #_w1;
   IF #_w3 THEN
       #H_SP3 := #MaxResSetp4 + 0.5;
       #H_SetpntAllowed := FALSE;
   END_IF;
END_REGION

REGION Network 48: **** 5.2 - Equations - Flow Equations **** Check Setpoint 4 with Setpoint 1 Resonance
   // Check Setpoint 4 with Setpoint 1 Resonance 
   // Setpoint 4 is no longer allowed, calculate prefered allowed setpoint 4
   // ENO of a box is taken as its EN; it also drops when the box reports an error
   #_w1 := (#SetpntChanged OR #SetpntBwdChanged OR #SetpntResChanged OR #CheckResSetpoints) AND (#H_SP4 <> 0.0) AND (#H_SP4 <= #MaxResSetp1) AND (#H_SP4 >= #MinResSetp1);
   #_w2 := (#H_SP4 <= #H_SPResonance1) AND #_w1;
   IF #_w2 THEN
       #H_SP4 := #MinResSetp1 - 0.5;
       #H_SetpntAllowed := FALSE;
   END_IF;
   #_w3 := (#H_SP4 > #H_SPResonance1) AND #_w1;
   IF #_w3 THEN
       #H_SP4 := #MaxResSetp1 + 0.5;
       #H_SetpntAllowed := FALSE;
   END_IF;
END_REGION

REGION Network 49: **** 5.2 - Equations - Flow Equations **** Check Setpoint 4 with Setpoint 2 Resonance
   // Check Setpoint 4 with Setpoint 2 Resonance 
   // Setpoint 4 is no longer allowed, calculate prefered allowed setpoint 4
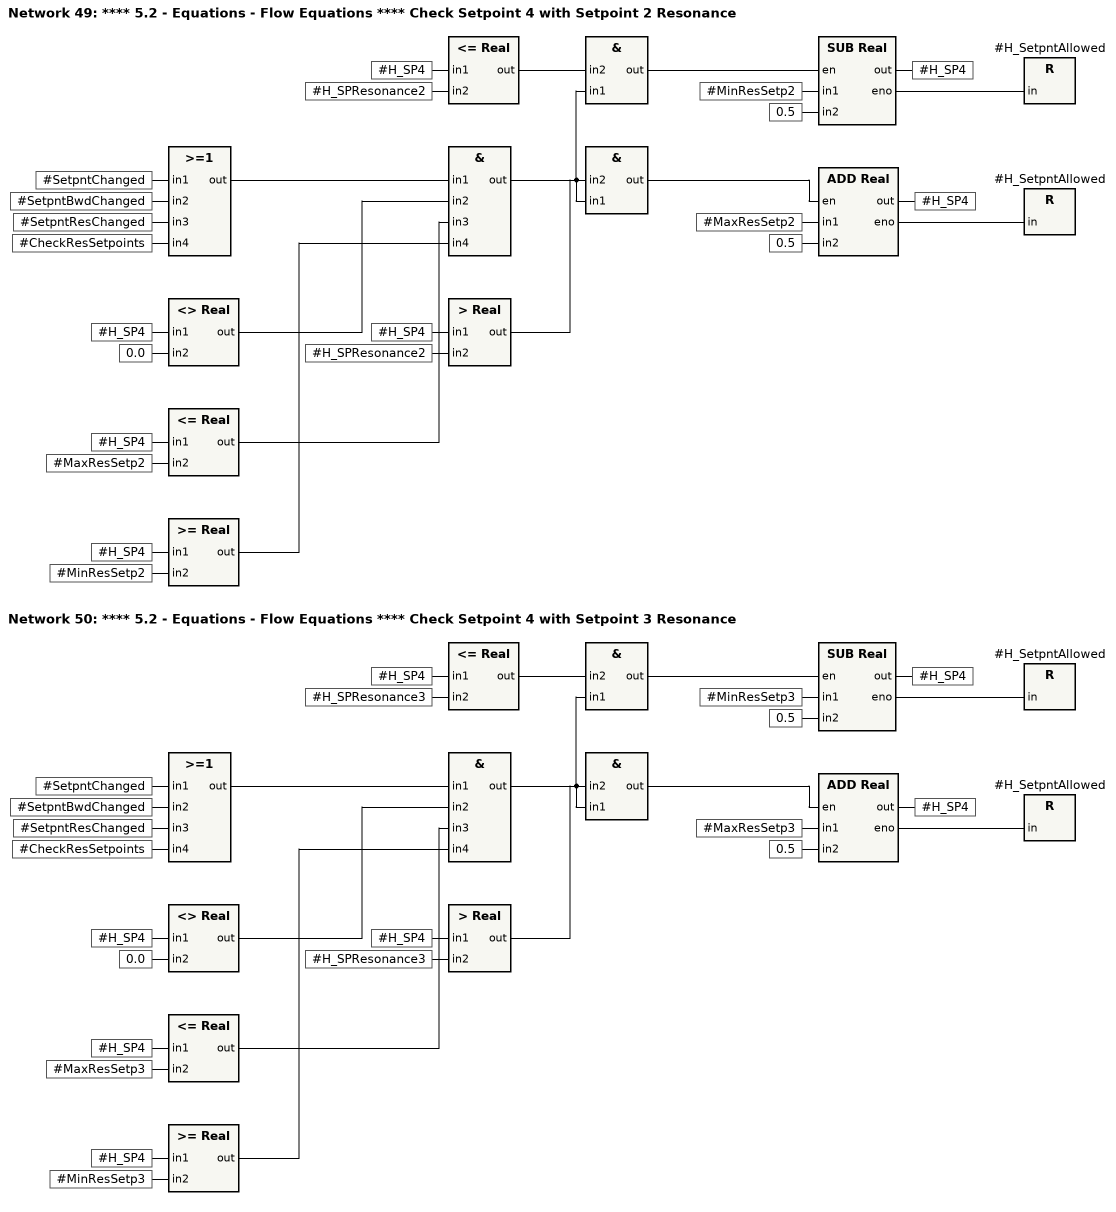
   // ENO of a box is taken as its EN; it also drops when the box reports an error
   #_w1 := (#SetpntChanged OR #SetpntBwdChanged OR #SetpntResChanged OR #CheckResSetpoints) AND (#H_SP4 <> 0.0) AND (#H_SP4 <= #MaxResSetp2) AND (#H_SP4 >= #MinResSetp2);
   #_w2 := (#H_SP4 <= #H_SPResonance2) AND #_w1;
   IF #_w2 THEN
       #H_SP4 := #MinResSetp2 - 0.5;
       #H_SetpntAllowed := FALSE;
   END_IF;
   #_w3 := (#H_SP4 > #H_SPResonance2) AND #_w1;
   IF #_w3 THEN
       #H_SP4 := #MaxResSetp2 + 0.5;
       #H_SetpntAllowed := FALSE;
   END_IF;
END_REGION

REGION Network 50: **** 5.2 - Equations - Flow Equations **** Check Setpoint 4 with Setpoint 3 Resonance
   // Check Setpoint 4 with Setpoint 3 Resonance 
   // Setpoint 4 is no longer allowed, calculate prefered allowed setpoint 4
   // ENO of a box is taken as its EN; it also drops when the box reports an error
   #_w1 := (#SetpntChanged OR #SetpntBwdChanged OR #SetpntResChanged OR #CheckResSetpoints) AND (#H_SP4 <> 0.0) AND (#H_SP4 <= #MaxResSetp3) AND (#H_SP4 >= #MinResSetp3);
   #_w2 := (#H_SP4 <= #H_SPResonance3) AND #_w1;
   IF #_w2 THEN
       #H_SP4 := #MinResSetp3 - 0.5;
       #H_SetpntAllowed := FALSE;
   END_IF;
   #_w3 := (#H_SP4 > #H_SPResonance3) AND #_w1;
   IF #_w3 THEN
       #H_SP4 := #MaxResSetp3 + 0.5;
       #H_SetpntAllowed := FALSE;
   END_IF;
END_REGION

REGION Network 51: **** 5.2 - Equations - Flow Equations **** Check Setpoint 4 with Setpoint 4 Resonance
   // Check Setpoint 4 with Setpoint 4 Resonance 
   // Setpoint 4 is no longer allowed, calculate prefered allowed setpoint 4
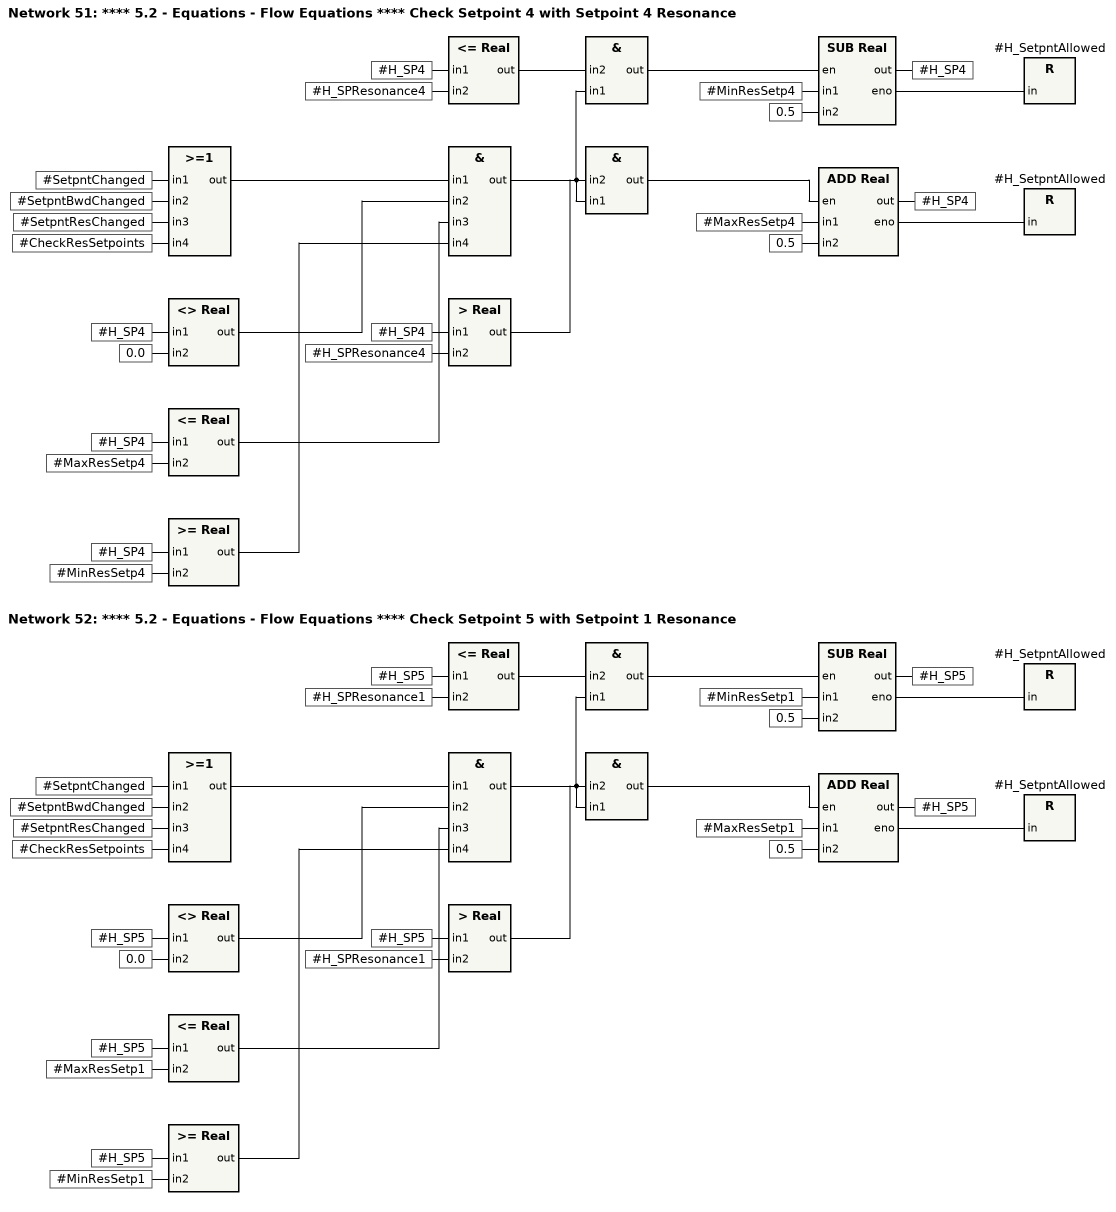
   // ENO of a box is taken as its EN; it also drops when the box reports an error
   #_w1 := (#SetpntChanged OR #SetpntBwdChanged OR #SetpntResChanged OR #CheckResSetpoints) AND (#H_SP4 <> 0.0) AND (#H_SP4 <= #MaxResSetp4) AND (#H_SP4 >= #MinResSetp4);
   #_w2 := (#H_SP4 <= #H_SPResonance4) AND #_w1;
   IF #_w2 THEN
       #H_SP4 := #MinResSetp4 - 0.5;
       #H_SetpntAllowed := FALSE;
   END_IF;
   #_w3 := (#H_SP4 > #H_SPResonance4) AND #_w1;
   IF #_w3 THEN
       #H_SP4 := #MaxResSetp4 + 0.5;
       #H_SetpntAllowed := FALSE;
   END_IF;
END_REGION

REGION Network 52: **** 5.2 - Equations - Flow Equations **** Check Setpoint 5 with Setpoint 1 Resonance
   // Check Setpoint 5 with Setpoint 1 Resonance 
   // Setpoint 5 is no longer allowed, calculate prefered allowed setpoint 5
   // ENO of a box is taken as its EN; it also drops when the box reports an error
   #_w1 := (#SetpntChanged OR #SetpntBwdChanged OR #SetpntResChanged OR #CheckResSetpoints) AND (#H_SP5 <> 0.0) AND (#H_SP5 <= #MaxResSetp1) AND (#H_SP5 >= #MinResSetp1);
   #_w2 := (#H_SP5 <= #H_SPResonance1) AND #_w1;
   IF #_w2 THEN
       #H_SP5 := #MinResSetp1 - 0.5;
       #H_SetpntAllowed := FALSE;
   END_IF;
   #_w3 := (#H_SP5 > #H_SPResonance1) AND #_w1;
   IF #_w3 THEN
       #H_SP5 := #MaxResSetp1 + 0.5;
       #H_SetpntAllowed := FALSE;
   END_IF;
END_REGION

REGION Network 53: **** 5.2 - Equations - Flow Equations ****Check Setpoint 5 with Setpoint 2 Resonance
   // Check Setpoint 5 with Setpoint 2 Resonance 
   // Setpoint 5 is no longer allowed, calculate prefered allowed setpoint 5
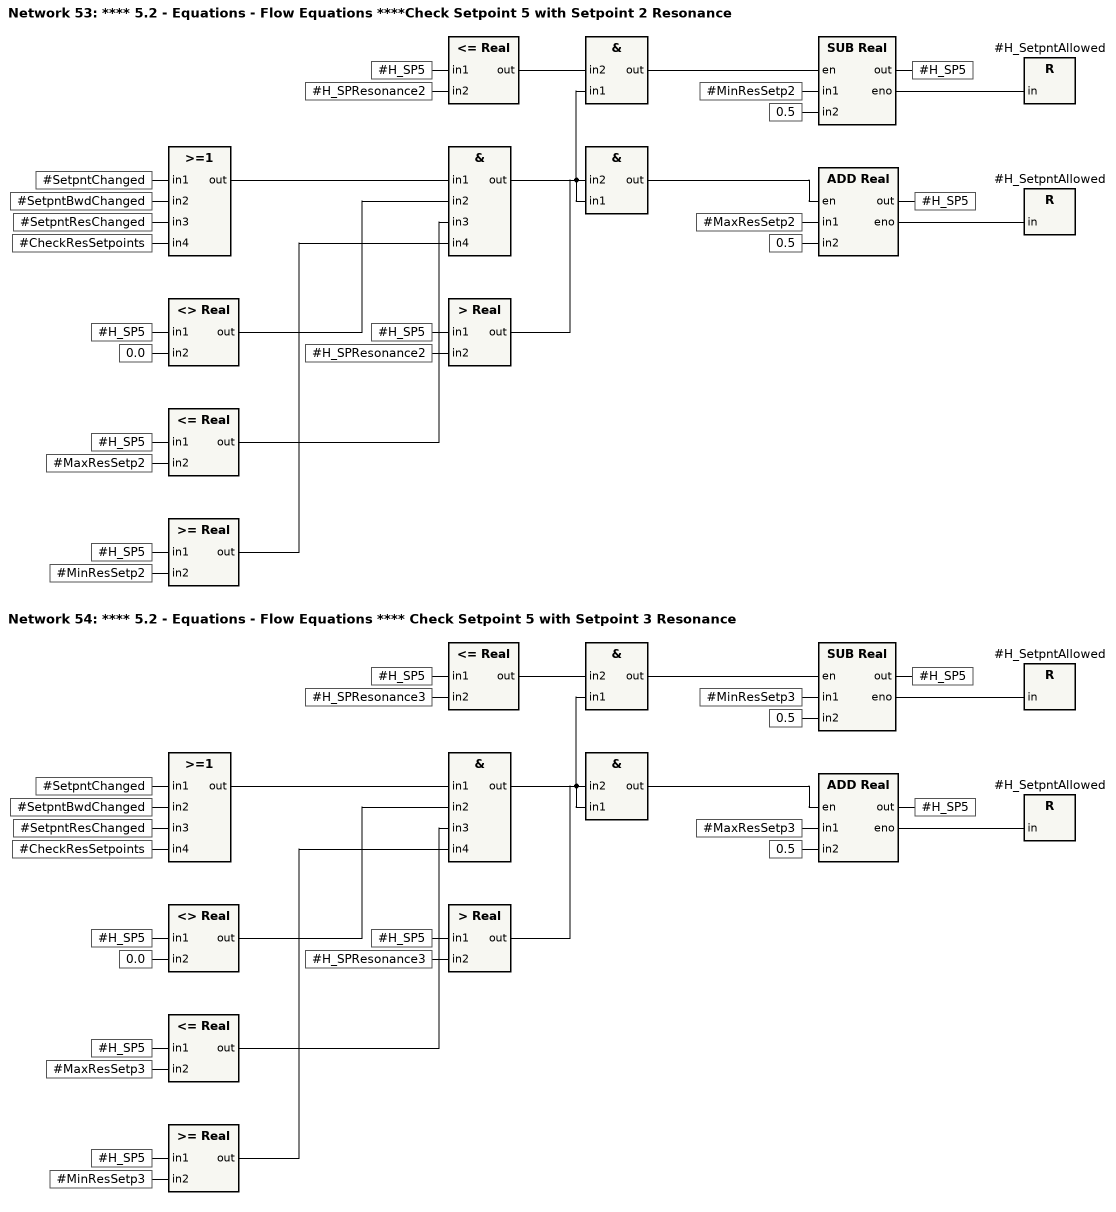
   // ENO of a box is taken as its EN; it also drops when the box reports an error
   #_w1 := (#SetpntChanged OR #SetpntBwdChanged OR #SetpntResChanged OR #CheckResSetpoints) AND (#H_SP5 <> 0.0) AND (#H_SP5 <= #MaxResSetp2) AND (#H_SP5 >= #MinResSetp2);
   #_w2 := (#H_SP5 <= #H_SPResonance2) AND #_w1;
   IF #_w2 THEN
       #H_SP5 := #MinResSetp2 - 0.5;
       #H_SetpntAllowed := FALSE;
   END_IF;
   #_w3 := (#H_SP5 > #H_SPResonance2) AND #_w1;
   IF #_w3 THEN
       #H_SP5 := #MaxResSetp2 + 0.5;
       #H_SetpntAllowed := FALSE;
   END_IF;
END_REGION

REGION Network 54: **** 5.2 - Equations - Flow Equations **** Check Setpoint 5 with Setpoint 3 Resonance
   // Check Setpoint 5 with Setpoint 3 Resonance 
   // Setpoint 5 is no longer allowed, calculate prefered allowed setpoint 5
   // ENO of a box is taken as its EN; it also drops when the box reports an error
   #_w1 := (#SetpntChanged OR #SetpntBwdChanged OR #SetpntResChanged OR #CheckResSetpoints) AND (#H_SP5 <> 0.0) AND (#H_SP5 <= #MaxResSetp3) AND (#H_SP5 >= #MinResSetp3);
   #_w2 := (#H_SP5 <= #H_SPResonance3) AND #_w1;
   IF #_w2 THEN
       #H_SP5 := #MinResSetp3 - 0.5;
       #H_SetpntAllowed := FALSE;
   END_IF;
   #_w3 := (#H_SP5 > #H_SPResonance3) AND #_w1;
   IF #_w3 THEN
       #H_SP5 := #MaxResSetp3 + 0.5;
       #H_SetpntAllowed := FALSE;
   END_IF;
END_REGION

REGION Network 55: **** 5.2 - Equations - Flow Equations **** Check Setpoint 5 with Setpoint 4 Resonance
   // Check Setpoint 5 with Setpoint 4 Resonance 
   // Setpoint 5 is no longer allowed, calculate prefered allowed setpoint 5
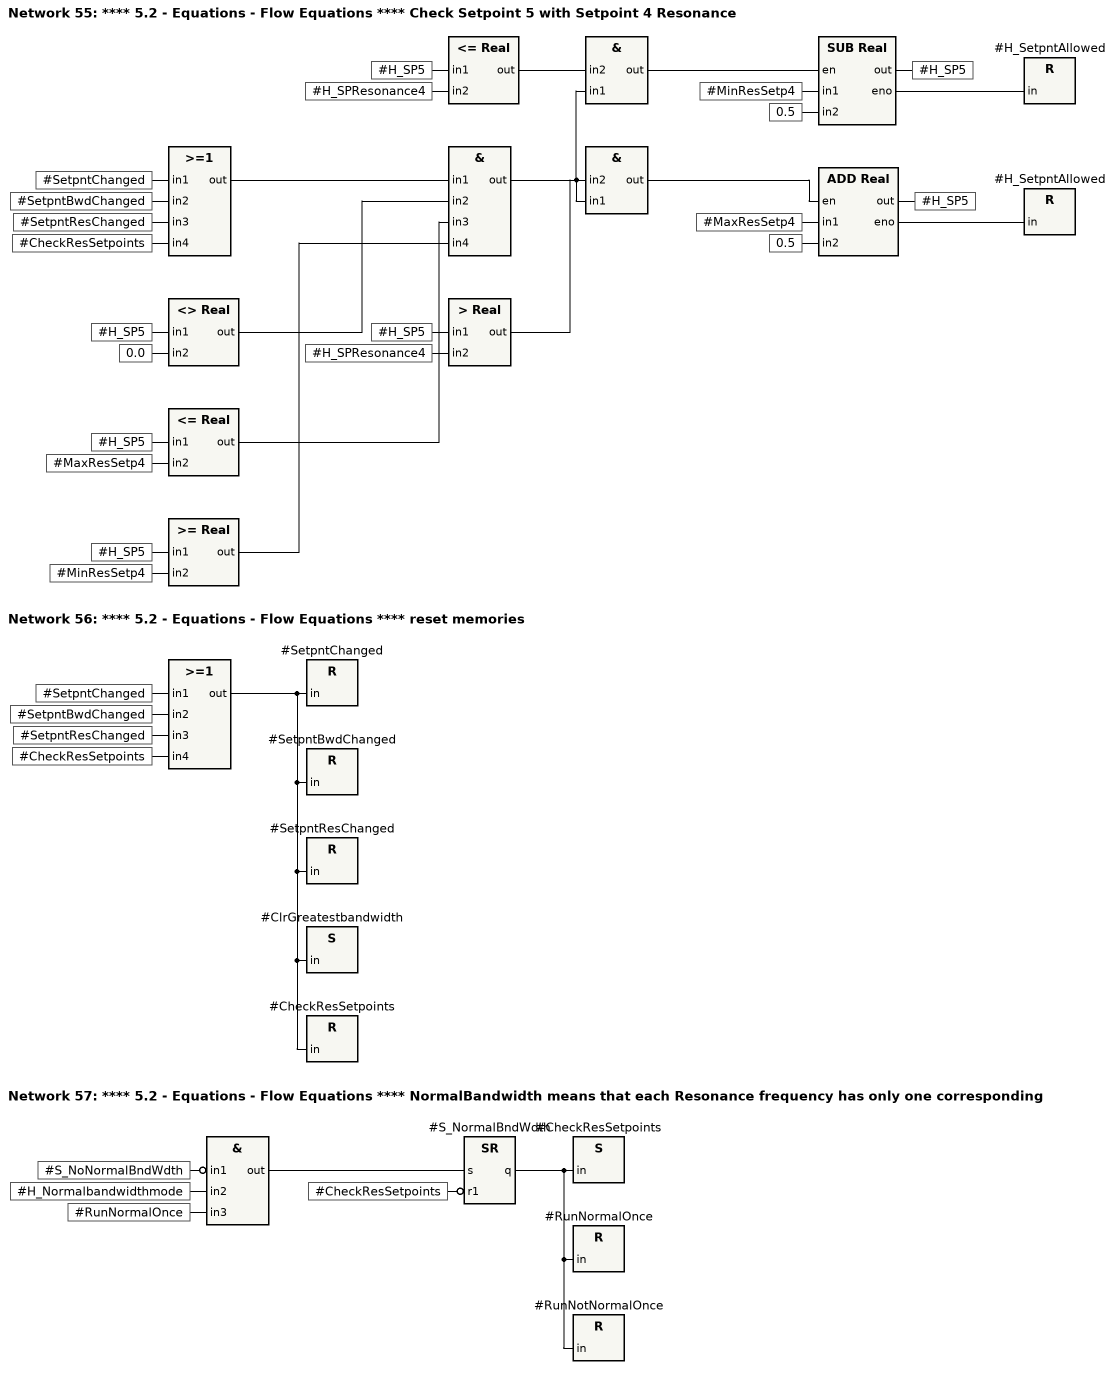
   // ENO of a box is taken as its EN; it also drops when the box reports an error
   #_w1 := (#SetpntChanged OR #SetpntBwdChanged OR #SetpntResChanged OR #CheckResSetpoints) AND (#H_SP5 <> 0.0) AND (#H_SP5 <= #MaxResSetp4) AND (#H_SP5 >= #MinResSetp4);
   #_w2 := (#H_SP5 <= #H_SPResonance4) AND #_w1;
   IF #_w2 THEN
       #H_SP5 := #MinResSetp4 - 0.5;
       #H_SetpntAllowed := FALSE;
   END_IF;
   #_w3 := (#H_SP5 > #H_SPResonance4) AND #_w1;
   IF #_w3 THEN
       #H_SP5 := #MaxResSetp4 + 0.5;
       #H_SetpntAllowed := FALSE;
   END_IF;
END_REGION

REGION Network 56: **** 5.2 - Equations - Flow Equations **** reset memories
   // reset memories
   #_w1 := #SetpntChanged OR #SetpntBwdChanged OR #SetpntResChanged OR #CheckResSetpoints;
   IF #_w1 THEN
       #SetpntChanged := FALSE;
       #SetpntBwdChanged := FALSE;
       #SetpntResChanged := FALSE;
       #ClrGreatestbandwidth := TRUE;
       #CheckResSetpoints := FALSE;
   END_IF;
END_REGION

REGION Network 57: **** 5.2 - Equations - Flow Equations **** NormalBandwidth means that each Resonance frequency has only one corresponding
   // NormalBandwidth means that each Resonance frequency has only one corresponding 
   // bandwidth
   IF NOT #S_NoNormalBndWdth AND #H_Normalbandwidthmode AND #RunNormalOnce THEN
       #S_NormalBndWdth := TRUE;   // SR flip-flop
   END_IF;
   IF NOT #CheckResSetpoints THEN #S_NormalBndWdth := FALSE; END_IF;
   IF #S_NormalBndWdth THEN
       #CheckResSetpoints := TRUE;
       #RunNormalOnce := FALSE;
       #RunNotNormalOnce := FALSE;
   END_IF;
END_REGION

REGION Network 58: **** 5.2 - Equations - Flow Equations **** Not NormalBandwidth means that each Resonance frequency works with the greatest
   // Not NormalBandwidth means that each Resonance frequency works with the greatest 
   // value of the 4 bandwidth's; it corresponds with the parametrizing of Danfoss 
   // frequency controller
   // bandwidth
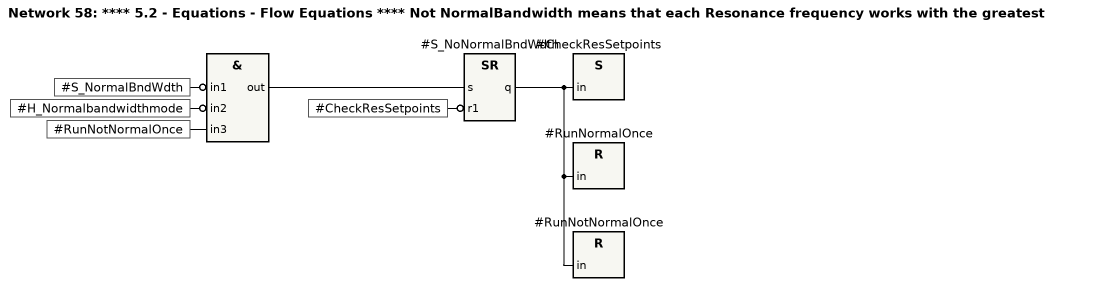
   IF NOT #S_NormalBndWdth AND NOT #H_Normalbandwidthmode AND #RunNotNormalOnce THEN
       #S_NoNormalBndWdth := TRUE;   // SR flip-flop
   END_IF;
   IF NOT #CheckResSetpoints THEN #S_NoNormalBndWdth := FALSE; END_IF;
   IF #S_NoNormalBndWdth THEN
       #CheckResSetpoints := TRUE;
       #RunNormalOnce := FALSE;
       #RunNotNormalOnce := FALSE;
   END_IF;
END_REGION
END_FUNCTION_BLOCK

FUNCTION_BLOCK "LProcDanfoss"   // FB1736, FBD
TITLE = LProcDanfoss
{ S7_Optimized_Access := 'FALSE' }
AUTHOR : VCC
FAMILY : ProcEq
NAME : DanfosDP
VERSION : 1.0
// ================================================================================
// Block to control a frequency controller Danfoss FC by Profinet or Profibus for 
// process applications.
// ================================================================================
// stored: AutoNumber false, IsIECCheckEnabled false, SetENOAutomatically False, UDAEnableTagReadback false
   VAR_INPUT
      I_EnableFCAlarm { ExternalAccessible := 'False'; ExternalVisible := 'False'; ExternalWritable := 'False'} : Bool;   // Enable alarm on frequency controller
      I_EnableCheckSpeedOK { ExternalAccessible := 'False'; ExternalVisible := 'False'; ExternalWritable := 'False'} : Bool;   // Enable check speed is OK
      I_EnableSafetySwitch { ExternalAccessible := 'False'; ExternalVisible := 'False'; ExternalWritable := 'False'} : Bool;   // Enable internal safety switch on drive
      I_AlarmResetPB { ExternalAccessible := 'False'; ExternalVisible := 'False'; ExternalWritable := 'False'} : Bool;   // Reset alarm from mode of station
      I_ReferenceValueLSB { ExternalAccessible := 'False'; ExternalVisible := 'False'; ExternalWritable := 'False'} : Bool;   // Control word to VLT : Reference value LSB
      I_ReferenceValueMSB { ExternalAccessible := 'False'; ExternalVisible := 'False'; ExternalWritable := 'False'} : Bool;   // Control word to VLT : Reference value MSB
      I_DCBrake { ExternalAccessible := 'False'; ExternalVisible := 'False'; ExternalWritable := 'False'} : Bool;   // Control word to VLT : DC Brake
      I_Coasting { ExternalAccessible := 'False'; ExternalVisible := 'False'; ExternalWritable := 'False'} : Bool;   // Control word to VLT : Coasting
      I_NotQuickStop { ExternalAccessible := 'False'; ExternalVisible := 'False'; ExternalWritable := 'False'} : Bool;   // Control word to VLT : Quick stop; When FALSE, the quickstop is active
      I_HoldOutputFreq { ExternalAccessible := 'False'; ExternalVisible := 'False'; ExternalWritable := 'False'} : Bool;   // Control word to VLT : Hold output frequency controller
      I_RampStopStart { ExternalAccessible := 'False'; ExternalVisible := 'False'; ExternalWritable := 'False'} : Bool;   // Control word to VLT : Ramp stop start
      I_Reset { ExternalAccessible := 'False'; ExternalVisible := 'False'; ExternalWritable := 'False'} : Bool;   // Control word to VLT : Reset
      I_Jog { ExternalAccessible := 'False'; ExternalVisible := 'False'; ExternalWritable := 'False'} : Bool;   // Control word to VLT : Jog function
      I_RampSelection { ExternalAccessible := 'False'; ExternalVisible := 'False'; ExternalWritable := 'False'} : Bool;   // Control word to VLT : Ramp selection
      I_DataValid { ExternalAccessible := 'False'; ExternalVisible := 'False'; ExternalWritable := 'False'} : Bool;   // Control word to VLT : Data Valid
      I_Relay01 { ExternalAccessible := 'False'; ExternalVisible := 'False'; ExternalWritable := 'False'} : Bool;   // Control word to VLT : Relay 01
      I_Relay04 { ExternalAccessible := 'False'; ExternalVisible := 'False'; ExternalWritable := 'False'} : Bool;   // Control word to VLT : Relay 04
      I_SetupSelectionLSB { ExternalAccessible := 'False'; ExternalVisible := 'False'; ExternalWritable := 'False'} : Bool;   // Control word to VLT : Setup Selection LSB
      I_SetupSelectionMSB { ExternalAccessible := 'False'; ExternalVisible := 'False'; ExternalWritable := 'False'} : Bool;   // Control word to VLT : Setup Selection MSB
      I_Reverse { ExternalAccessible := 'False'; ExternalVisible := 'False'; ExternalWritable := 'False'} : Bool;   // Control word to VLT : Reverse
      I_HWSubInput { ExternalAccessible := 'False'; ExternalVisible := 'False'; ExternalWritable := 'False'} : HW_SUBMODULE;   // I/O connection hardware
      I_HWSubOutput { ExternalAccessible := 'False'; ExternalVisible := 'False'; ExternalWritable := 'False'} : HW_SUBMODULE;   // I/O connection hardware
      I_MRV_FC { ExternalAccessible := 'False'; ExternalVisible := 'False'; ExternalWritable := 'False'} : Int;   // Speed reference (% of max reference)
      I_PCDIndex1 { ExternalAccessible := 'False'; ExternalVisible := 'False'; ExternalWritable := 'False'} : Int;   // PCD index 1 value
      I_PCDIndex2 { ExternalAccessible := 'False'; ExternalVisible := 'False'; ExternalWritable := 'False'} : Int;   // PCD index 2 value
      I_PCDIndex3 { ExternalAccessible := 'False'; ExternalVisible := 'False'; ExternalWritable := 'False'} : Int;   // PCD index 3 value
      I_PCDIndex4 { ExternalAccessible := 'False'; ExternalVisible := 'False'; ExternalWritable := 'False'} : Int;   // PCD index 4 value
      I_PCDIndex5 { ExternalAccessible := 'False'; ExternalVisible := 'False'; ExternalWritable := 'False'} : Int;   // PCD index 5 value
      I_PCDIndex6 { ExternalAccessible := 'False'; ExternalVisible := 'False'; ExternalWritable := 'False'} : Int;   // PCD index 6 value
      I_PCDIndex7 { ExternalAccessible := 'False'; ExternalVisible := 'False'; ExternalWritable := 'False'} : Int;   // PCD index 7 value
      I_PCDIndex8 { ExternalAccessible := 'False'; ExternalVisible := 'False'; ExternalWritable := 'False'} : Int;   // PCD index 8 value
      I_TimeCheckSpeedOK { ExternalAccessible := 'False'; ExternalVisible := 'False'; ExternalWritable := 'False'} : DInt;   // Delay time to check if speed is OK
   END_VAR
   VAR_OUTPUT
      O_FCAlarm { ExternalAccessible := 'False'; ExternalVisible := 'False'; ExternalWritable := 'False'} : Bool;   // Frequency controller is in alarm
      O_FCAlarmC { ExternalAccessible := 'False'; ExternalVisible := 'False'; ExternalWritable := 'False'} : Bool;   // Frequency controller is in alarm C
      O_AlarmABCondition { ExternalAccessible := 'False'; ExternalVisible := 'False'; ExternalWritable := 'False'} : Bool;   // Alarm AB condition
      O_Active { ExternalAccessible := 'False'; ExternalVisible := 'False'; ExternalWritable := 'False'} : Bool;   // Frequency controller - Profibus active
      H_IAnim { ExternalAccessible := 'False'; ExternalVisible := 'False'; ExternalWritable := 'False'} : Word;   // HMI Animation color of the icon
   END_VAR
   VAR DB_SPECIFIC
      H_Out : Struct   // HMI
         Anim : Word;   // HMI Animation of the object
         FromFC_STW : Int;   // HMI Animation: Value of STW (status word)
         FromFC_MAV : Int;   // HMI Animation: Value of main reference (real speed)
         FromFC_Index1 : Int;   // HMI Animation: Value of Index 1
         FromFC_Index2 : Int;   // HMI Animation: Value of Index 2
         FromFC_Index3 : Int;   // HMI Animation: Value of Index 3
         FromFC_Index4 : Int;   // HMI Animation: Value of Index 4
         FromFC_Index5 : Int;   // HMI Animation: Value of Index 5
         FromFC_Index6 : Int;   // HMI Animation: Value of Index 6
         FromFC_Index7 : Int;   // HMI Animation: Value of Index 7
         FromFC_Index8 : Int;   // HMI Animation: Value of Index 8
         ToFC_CTW : Int;   // HMI Animation: Value of CTW (control word)
         ToFC_MRV : Int;   // HMI Animation: Value of MRV (speed setup)
         DBnr : Int;   // HMI Animation DB number
      END_STRUCT;
      FCAlarmA { ExternalAccessible := 'False'; ExternalVisible := 'False'; ExternalWritable := 'False'} : Bool;   // Frequency controller is in alarm A
      FCAlarmC { ExternalAccessible := 'False'; ExternalVisible := 'False'; ExternalWritable := 'False'} : Bool;   // Frequency controller is in alarm C
      FCAlarmAlmCond { ExternalAccessible := 'False'; ExternalVisible := 'False'; ExternalWritable := 'False'} : Bool;   // Frequency controller alarm condition
      Active { ExternalAccessible := 'False'; ExternalVisible := 'False'; ExternalWritable := 'False'} : Bool;   // Frequency controller - Profibus active
      CheckSpeedOK { ExternalAccessible := 'False'; ExternalVisible := 'False'; ExternalWritable := 'False'} : Bool;   // Check speed OK alarm for internal diagnostic use
      SpeedOKAlm { ExternalAccessible := 'False'; ExternalVisible := 'False'; ExternalWritable := 'False'} : Bool;   // Speed OK alarm for internal diagnostic use
      BusControlAlm { ExternalAccessible := 'False'; ExternalVisible := 'False'; ExternalWritable := 'False'} : Bool;   // Bus control alarm for internal diagnostic use
      AutostartAlm { ExternalAccessible := 'False'; ExternalVisible := 'False'; ExternalWritable := 'False'} : Bool;   // AutostartAlm alarm for internal diagnostic use
      TripAlm { ExternalAccessible := 'False'; ExternalVisible := 'False'; ExternalWritable := 'False'} : Bool;   // Trip alarm for internal diagnostic use
      ErrorAlm { ExternalAccessible := 'False'; ExternalVisible := 'False'; ExternalWritable := 'False'} : Bool;   // Error but not trip alarm for internal diagnostic use
      TripLockAlm { ExternalAccessible := 'False'; ExternalVisible := 'False'; ExternalWritable := 'False'} : Bool;   // Trip and lock alarm for internal diagnostic use
      SafetySwitchAlm { ExternalAccessible := 'False'; ExternalVisible := 'False'; ExternalWritable := 'False'} : Bool;   // Safety switch alarm for internal diagnostic use
      WarningAlm { ExternalAccessible := 'False'; ExternalVisible := 'False'; ExternalWritable := 'False'} : Bool;   // Warning alarm for internal diagnostic use
      VoltageLimitExceedAlm { ExternalAccessible := 'False'; ExternalVisible := 'False'; ExternalWritable := 'False'} : Bool;   // Voltage too high or too low alarm for internal diagnostic use
      TorqueLimitExceedAlm { ExternalAccessible := 'False'; ExternalVisible := 'False'; ExternalWritable := 'False'} : Bool;   // Torque too high or too low alarm for internal diagnostic use
      TimerLimitExceedAlm { ExternalAccessible := 'False'; ExternalVisible := 'False'; ExternalWritable := 'False'} : Bool;   // Timer overtemperature alarm for internal diagnostic use
      FrequencyLimitAlm { ExternalAccessible := 'False'; ExternalVisible := 'False'; ExternalWritable := 'False'} : Bool;   // Frequency limit alarm for internal diagnostic use
      HeatsinkTempAlm { ExternalAccessible := 'False'; ExternalVisible := 'False'; ExternalWritable := 'False'} : Bool;   // Heatsink temperature alarm for internal diagnostic use
      RetValueDataFromFC { ExternalAccessible := 'False'; ExternalVisible := 'False'; ExternalWritable := 'False'} : Int;   // Status variable (SFC14)
      RetValueDataToFC { ExternalAccessible := 'False'; ExternalVisible := 'False'; ExternalWritable := 'False'} : Int;   // Status variable (SFC15)
      DBnr { ExternalAccessible := 'False'; ExternalVisible := 'False'; ExternalWritable := 'False'} : Int;   // HMI DB number
   END_VAR
   VAR
      SpeedOKTimer { ExternalAccessible := 'False'; ExternalVisible := 'False'; ExternalWritable := 'False'; S7_SetPoint := 'True'} : "LTimer";   // Timer check speed is OK
      STW_Alarm { ExternalAccessible := 'False'; ExternalVisible := 'False'; ExternalWritable := 'False'; S7_SetPoint := 'True'} : "LProc1AlarmMultiIn";   // Alarms fequency controller
      DelayAlarmC { ExternalAccessible := 'False'; ExternalVisible := 'False'; ExternalWritable := 'False'; S7_SetPoint := 'True'} : "LTimer";   // Timer Delay Alarm C
   END_VAR
   VAR DB_SPECIFIC
      DataFromFC { ExternalAccessible := 'False'; ExternalVisible := 'False'; ExternalWritable := 'False'} : Struct   // Temp structure : receive data's from Frequency controller
         STW { ExternalAccessible := 'False'; ExternalVisible := 'False'; ExternalWritable := 'False'} : Struct   // From FC : STW (stat word)
            SpeedOK { ExternalAccessible := 'False'; ExternalVisible := 'False'; ExternalWritable := 'False'} : Bool;   // Status word from FC : Speed is OK
            BusControl { ExternalAccessible := 'False'; ExternalVisible := 'False'; ExternalWritable := 'False'} : Bool;   // Status word from FC : Frequency controller can be controlled via fieldbus
            FrequencyLimit { ExternalAccessible := 'False'; ExternalVisible := 'False'; ExternalWritable := 'False'} : Bool;   // Status word from FC : Frequency output within the defined limits
            InOperation { ExternalAccessible := 'False'; ExternalVisible := 'False'; ExternalWritable := 'False'} : Bool;   // Status word from FC : Frequency controller started (freq > 0 Hz)
            Autostart { ExternalAccessible := 'False'; ExternalVisible := 'False'; ExternalWritable := 'False'} : Bool;   // Status word from FC : Frequency controller start due to over temperature
            VoltageLimitExceed { ExternalAccessible := 'False'; ExternalVisible := 'False'; ExternalWritable := 'False'} : Bool;   // Status word from FC : Frequency controller voltage is too low or too high
            TorqueLimitExceed { ExternalAccessible := 'False'; ExternalVisible := 'False'; ExternalWritable := 'False'} : Bool;   // Status word from FC : Frequency controller torque is too low or too high
            TimerLimitExceed { ExternalAccessible := 'False'; ExternalVisible := 'False'; ExternalWritable := 'False'} : Bool;   // Status word from FC : Frequency controller timer over temp on motor or VLT
            FCReady { ExternalAccessible := 'False'; ExternalVisible := 'False'; ExternalWritable := 'False'} : Bool;   // Status word from FC : Frequency controller ready
            DriveReady { ExternalAccessible := 'False'; ExternalVisible := 'False'; ExternalWritable := 'False'} : Bool;   // Status word from FC : Frequency controller ready for operation
            CostingStop { ExternalAccessible := 'False'; ExternalVisible := 'False'; ExternalWritable := 'False'} : Bool;   // Status word from FC : Frequency controller can start the motor
            Trip { ExternalAccessible := 'False'; ExternalVisible := 'False'; ExternalWritable := 'False'} : Bool;   // Status word from FC : Frequency controller tripped
            Error { ExternalAccessible := 'False'; ExternalVisible := 'False'; ExternalWritable := 'False'} : Bool;   // Status word from FC : Frequency controller error but not trip
            NotUsed { ExternalAccessible := 'False'; ExternalVisible := 'False'; ExternalWritable := 'False'} : Bool;   // Status word from FC : not used
            TripLock { ExternalAccessible := 'False'; ExternalVisible := 'False'; ExternalWritable := 'False'} : Bool;   // Status word from FC : Frequency controller trip and lock
            Warning { ExternalAccessible := 'False'; ExternalVisible := 'False'; ExternalWritable := 'False'} : Bool;   // Status word from FC : Warning has occured
         END_STRUCT;
         MAV { ExternalAccessible := 'False'; ExternalVisible := 'False'; ExternalWritable := 'False'} : Int;   // From FC : MAV (actual main reference from Frequency controller)
         PCDIndex1Value { ExternalAccessible := 'False'; ExternalVisible := 'False'; ExternalWritable := 'False'} : Int;   // From FC : Value of PCD Index 1
         PCDIndex2Value { ExternalAccessible := 'False'; ExternalVisible := 'False'; ExternalWritable := 'False'} : Int;   // From FC : Value of PCD Index 2
         PCDIndex3Value { ExternalAccessible := 'False'; ExternalVisible := 'False'; ExternalWritable := 'False'} : Int;   // From FC : Value of PCD Index 3
         PCDIndex4Value { ExternalAccessible := 'False'; ExternalVisible := 'False'; ExternalWritable := 'False'} : Int;   // From FC : Value of PCD Index 4
         PCDIndex5Value { ExternalAccessible := 'False'; ExternalVisible := 'False'; ExternalWritable := 'False'} : Int;   // From FC : Value of PCD Index 5
         PCDIndex6Value { ExternalAccessible := 'False'; ExternalVisible := 'False'; ExternalWritable := 'False'} : Int;   // From FC : Value of PCD Index 6
         PCDIndex7Value { ExternalAccessible := 'False'; ExternalVisible := 'False'; ExternalWritable := 'False'} : Int;   // From FC : Value of PCD Index 7
         PCDIndex8Value { ExternalAccessible := 'False'; ExternalVisible := 'False'; ExternalWritable := 'False'} : Int;   // From FC : Value of PCD Index 8
      END_STRUCT;
      DataToFC { ExternalAccessible := 'False'; ExternalVisible := 'False'; ExternalWritable := 'False'} : Struct   // Temp structure : deliver data's to Frequency controller
         CTW { ExternalAccessible := 'False'; ExternalVisible := 'False'; ExternalWritable := 'False'} : Struct   // To FC : CTW (control word)
            Jog { ExternalAccessible := 'False'; ExternalVisible := 'False'; ExternalWritable := 'False'} : Bool;   // Control word to FC : Jog function
            RampSelection { ExternalAccessible := 'False'; ExternalVisible := 'False'; ExternalWritable := 'False'} : Bool;   // Control word to FC : Ramp selection
            DataValid { ExternalAccessible := 'False'; ExternalVisible := 'False'; ExternalWritable := 'False'} : Bool;   // Control word to FC : Data Valid
            Relay01 { ExternalAccessible := 'False'; ExternalVisible := 'False'; ExternalWritable := 'False'} : Bool;   // Control word to FC : Relay 01
            Relay04 { ExternalAccessible := 'False'; ExternalVisible := 'False'; ExternalWritable := 'False'} : Bool;   // Control word to FC : Relay 04
            SetupSelectionLSB { ExternalAccessible := 'False'; ExternalVisible := 'False'; ExternalWritable := 'False'} : Bool;   // Control word to FC : Setup selection LSB
            SetupSelectionMSB { ExternalAccessible := 'False'; ExternalVisible := 'False'; ExternalWritable := 'False'} : Bool;   // Control word to FC : Setup selection MSB
            Reverse { ExternalAccessible := 'False'; ExternalVisible := 'False'; ExternalWritable := 'False'} : Bool;   // Control word to FC : Reverse
            ReferenceValueLSB { ExternalAccessible := 'False'; ExternalVisible := 'False'; ExternalWritable := 'False'} : Bool;   // Control word to FC : Reference Value LSB
            ReferenceValueMSB { ExternalAccessible := 'False'; ExternalVisible := 'False'; ExternalWritable := 'False'} : Bool;   // Control word to FC : Reference Value MSB
            DCBrake { ExternalAccessible := 'False'; ExternalVisible := 'False'; ExternalWritable := 'False'} : Bool;   // Control word to FC : DC Brake
            Coasting { ExternalAccessible := 'False'; ExternalVisible := 'False'; ExternalWritable := 'False'} : Bool;   // Control word to FC : Coasting
            QuickStop { ExternalAccessible := 'False'; ExternalVisible := 'False'; ExternalWritable := 'False'} : Bool;   // Control word to FC : Quick Stop
            HoldOutputFreq { ExternalAccessible := 'False'; ExternalVisible := 'False'; ExternalWritable := 'False'} : Bool;   // Control word to FC : Hold output frequency controller
            RampStopStart { ExternalAccessible := 'False'; ExternalVisible := 'False'; ExternalWritable := 'False'} : Bool;   // Control word to FC : Ramp Stop Start
            Reset { ExternalAccessible := 'False'; ExternalVisible := 'False'; ExternalWritable := 'False'} : Bool;   // Control word to FC : Reset
         END_STRUCT;
         MRV { ExternalAccessible := 'False'; ExternalVisible := 'False'; ExternalWritable := 'False'} : Int;   // To FC : Main reference (setup)
         PCDIndex1 { ExternalAccessible := 'False'; ExternalVisible := 'False'; ExternalWritable := 'False'} : Int;   // To FC : PCD Index 1
         PCDIndex2 { ExternalAccessible := 'False'; ExternalVisible := 'False'; ExternalWritable := 'False'} : Int;   // To FC : PCD Index 2
         PCDIndex3 { ExternalAccessible := 'False'; ExternalVisible := 'False'; ExternalWritable := 'False'} : Int;   // To FC : PCD Index 3
         PCDIndex4 { ExternalAccessible := 'False'; ExternalVisible := 'False'; ExternalWritable := 'False'} : Int;   // To FC : PCD Index 4
         PCDIndex5 { ExternalAccessible := 'False'; ExternalVisible := 'False'; ExternalWritable := 'False'} : Int;   // To FC : PCD Index 5
         PCDIndex6 { ExternalAccessible := 'False'; ExternalVisible := 'False'; ExternalWritable := 'False'} : Int;   // To FC : PCD Index 6
         PCDIndex7 { ExternalAccessible := 'False'; ExternalVisible := 'False'; ExternalWritable := 'False'} : Int;   // To FC : PCD Index 7
         PCDIndex8 { ExternalAccessible := 'False'; ExternalVisible := 'False'; ExternalWritable := 'False'} : Int;   // To FC : PCD Index 8
      END_STRUCT;
      SafetySwitch { ExternalAccessible := 'False'; ExternalVisible := 'False'; ExternalWritable := 'False'} : Bool;   // Temp safety switch input from Frequency controller
      MRV_FC_Real { ExternalAccessible := 'False'; ExternalVisible := 'False'; ExternalWritable := 'False'} : Real;   // Temp Speed reference (% of max reference) as real
      MRV_FC_Dec { ExternalAccessible := 'False'; ExternalVisible := 'False'; ExternalWritable := 'False'} : Real;   // Temp Speed reference (decimal of max reference)
      MRV_FC_DInt { ExternalAccessible := 'False'; ExternalVisible := 'False'; ExternalWritable := 'False'} : DInt;   // Temp Speed reference (decimal of max reference) as DInt
   END_VAR
BEGIN

NETWORK
TITLE = **** 1 - Inputs **** DB number
// DB number
      L     DINO;
      T     #DBnr;

REGION Network 2: **** 1 - Inputs **** Profibus communication
   // Profibus communication
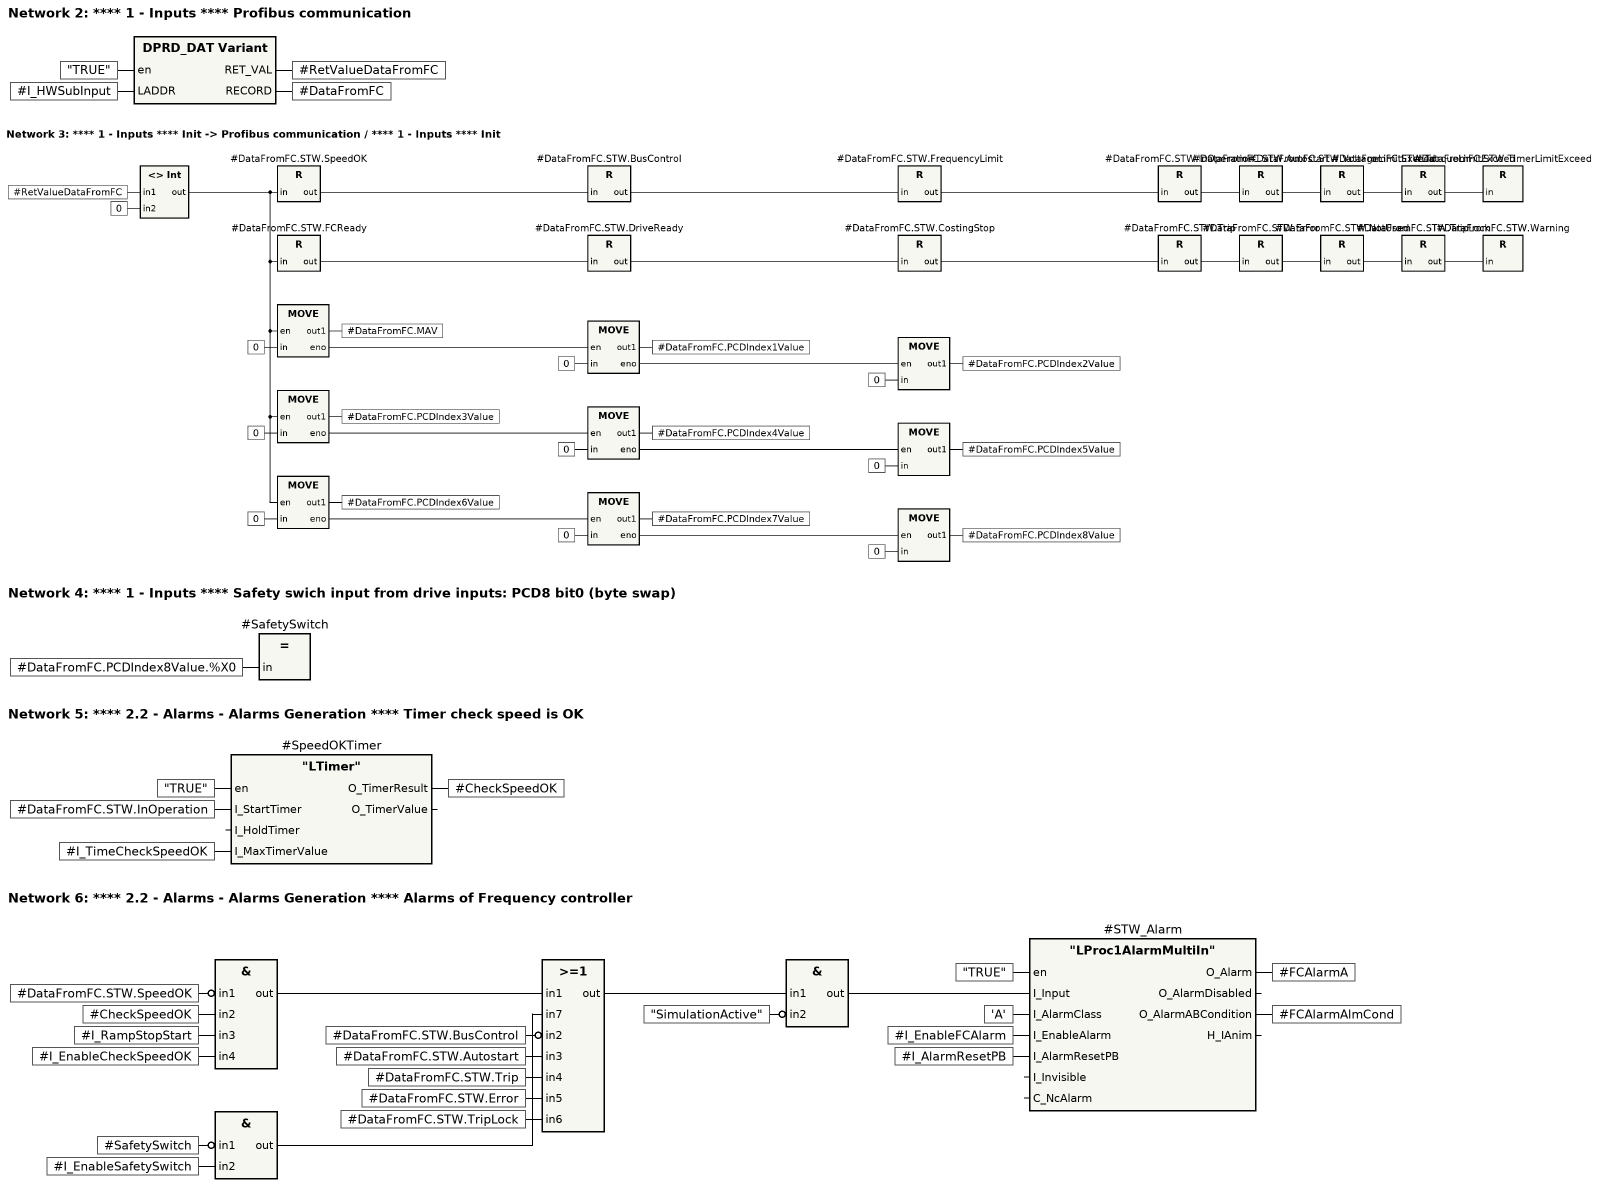
   IF "TRUE" THEN #RetValueDataFromFC := DPRD_DAT(LADDR := #I_HWSubInput, RECORD => #DataFromFC); END_IF;
END_REGION

REGION Network 3: **** 1 - Inputs **** Init -> Profibus communication / **** 1 - Inputs **** Init
   // Init -> Profibus communication / Init
   IF #RetValueDataFromFC <> 0 THEN
       #DataFromFC.STW.SpeedOK := FALSE;
       #DataFromFC.STW.BusControl := FALSE;
       #DataFromFC.STW.FrequencyLimit := FALSE;
       #DataFromFC.STW.InOperation := FALSE;
       #DataFromFC.STW.Autostart := FALSE;
       #DataFromFC.STW.VoltageLimitExceed := FALSE;
       #DataFromFC.STW.TorqueLimitExceed := FALSE;
       #DataFromFC.STW.TimerLimitExceed := FALSE;
       #DataFromFC.STW.FCReady := FALSE;
       #DataFromFC.STW.DriveReady := FALSE;
       #DataFromFC.STW.CostingStop := FALSE;
       #DataFromFC.STW.Trip := FALSE;
       #DataFromFC.STW.Error := FALSE;
       #DataFromFC.STW.NotUsed := FALSE;
       #DataFromFC.STW.TripLock := FALSE;
       #DataFromFC.STW.Warning := FALSE;
       #DataFromFC.MAV := 0;
       #DataFromFC.PCDIndex1Value := 0;
       #DataFromFC.PCDIndex2Value := 0;
       #DataFromFC.PCDIndex3Value := 0;
       #DataFromFC.PCDIndex4Value := 0;
       #DataFromFC.PCDIndex5Value := 0;
       #DataFromFC.PCDIndex6Value := 0;
       #DataFromFC.PCDIndex7Value := 0;
       #DataFromFC.PCDIndex8Value := 0;
   END_IF;
END_REGION

REGION Network 4: **** 1 - Inputs **** Safety swich input from drive inputs: PCD8 bit0 (byte swap)
   // Safety swich input from drive inputs: PCD8 bit0 (byte swap)
   #SafetySwitch := #DataFromFC.PCDIndex8Value.%X0;
END_REGION

REGION Network 5: **** 2.2 - Alarms - Alarms Generation **** Timer check speed is OK
   // Timer check speed is OK
   IF "TRUE" THEN
       #SpeedOKTimer(I_StartTimer := #DataFromFC.STW.InOperation,   // "LTimer"
                     I_MaxTimerValue := #I_TimeCheckSpeedOK,
                     O_TimerResult => #CheckSpeedOK);
   END_IF;
END_REGION

REGION Network 6: **** 2.2 - Alarms - Alarms Generation **** Alarms of Frequency controller
   // Alarms of Frequency controller
   IF "TRUE" THEN
       #STW_Alarm(I_Input := ((NOT #DataFromFC.STW.SpeedOK AND #CheckSpeedOK AND #I_RampStopStart AND #I_EnableCheckSpeedOK) OR (NOT #SafetySwitch AND #I_EnableSafetySwitch) OR NOT #DataFromFC.STW.BusControl OR #DataFromFC.STW.Autostart OR #DataFromFC.STW.Trip OR #DataFromFC.STW.Error OR #DataFromFC.STW.TripLock) AND NOT "SimulationActive",   // "LProc1AlarmMultiIn"
                  I_AlarmClass := 'A',
                  I_EnableAlarm := #I_EnableFCAlarm,
                  I_AlarmResetPB := #I_AlarmResetPB,
                  O_Alarm => #FCAlarmA,
                  O_AlarmABCondition => #FCAlarmAlmCond);
   END_IF;
END_REGION

REGION Network 7: **** 2.2 - Alarms - Alarms Generation **** Alarms C of Frequency controller
   // Alarms C of Frequency controller
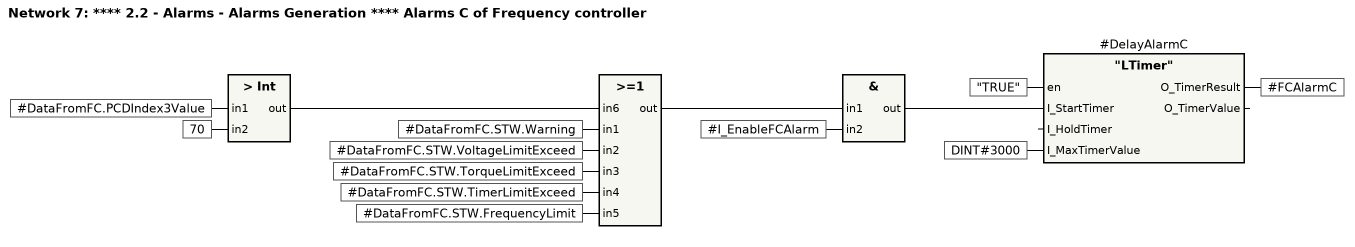
   IF "TRUE" THEN
       #DelayAlarmC(I_StartTimer := ((#DataFromFC.PCDIndex3Value > 70) OR #DataFromFC.STW.Warning OR #DataFromFC.STW.VoltageLimitExceed OR #DataFromFC.STW.TorqueLimitExceed OR #DataFromFC.STW.TimerLimitExceed OR #DataFromFC.STW.FrequencyLimit) AND #I_EnableFCAlarm,   // "LTimer"
                    I_MaxTimerValue := DINT#3000,
                    O_TimerResult => #FCAlarmC);
   END_IF;
END_REGION

REGION Network 8: **** 2.2 - Alarms - Alarms Generation **** Generate individual alarms for alarms from frequency converter
   // Generate individual alarms for alarms from frequency converter
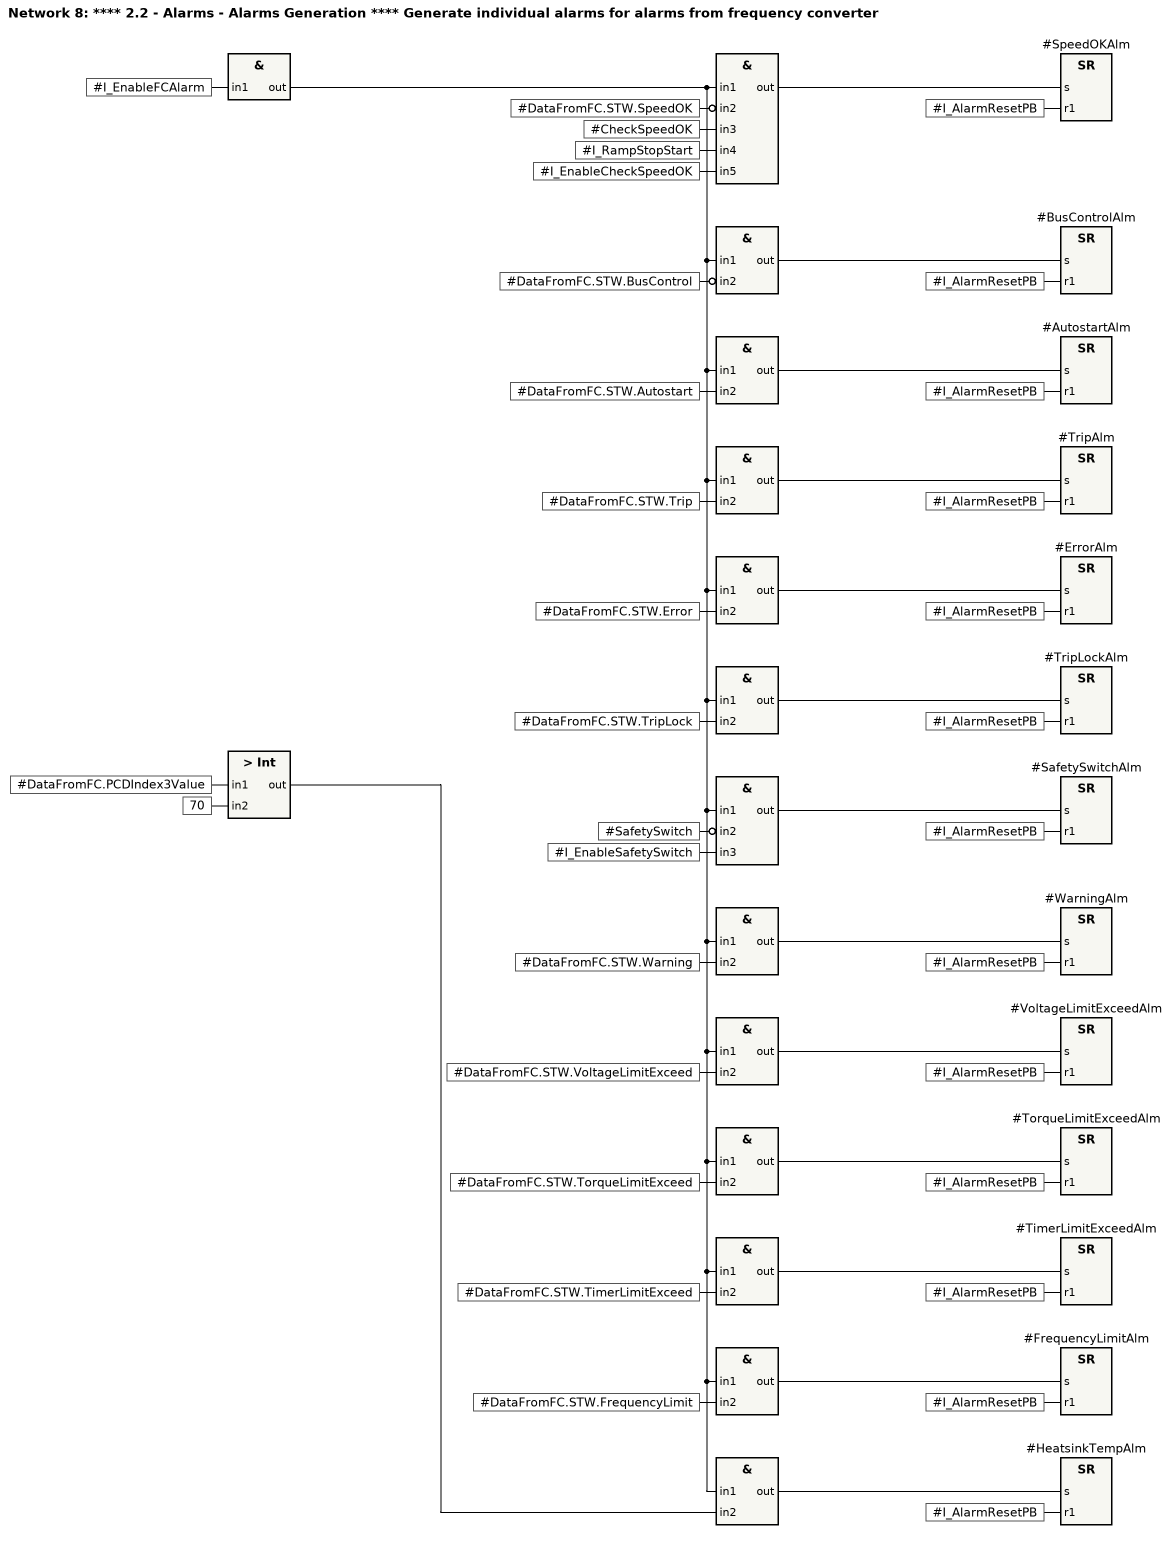
   IF #I_EnableFCAlarm AND NOT #DataFromFC.STW.SpeedOK AND #CheckSpeedOK AND #I_RampStopStart AND #I_EnableCheckSpeedOK THEN
       #SpeedOKAlm := TRUE;   // SR flip-flop
   END_IF;
   IF #I_AlarmResetPB THEN #SpeedOKAlm := FALSE; END_IF;
   IF #I_EnableFCAlarm AND NOT #DataFromFC.STW.BusControl THEN
       #BusControlAlm := TRUE;   // SR flip-flop
   END_IF;
   IF #I_AlarmResetPB THEN #BusControlAlm := FALSE; END_IF;
   IF #I_EnableFCAlarm AND #DataFromFC.STW.Autostart THEN
       #AutostartAlm := TRUE;   // SR flip-flop
   END_IF;
   IF #I_AlarmResetPB THEN #AutostartAlm := FALSE; END_IF;
   IF #I_EnableFCAlarm AND #DataFromFC.STW.Trip THEN
       #TripAlm := TRUE;   // SR flip-flop
   END_IF;
   IF #I_AlarmResetPB THEN #TripAlm := FALSE; END_IF;
   IF #I_EnableFCAlarm AND #DataFromFC.STW.Error THEN
       #ErrorAlm := TRUE;   // SR flip-flop
   END_IF;
   IF #I_AlarmResetPB THEN #ErrorAlm := FALSE; END_IF;
   IF #I_EnableFCAlarm AND #DataFromFC.STW.TripLock THEN
       #TripLockAlm := TRUE;   // SR flip-flop
   END_IF;
   IF #I_AlarmResetPB THEN #TripLockAlm := FALSE; END_IF;
   IF #I_EnableFCAlarm AND NOT #SafetySwitch AND #I_EnableSafetySwitch THEN
       #SafetySwitchAlm := TRUE;   // SR flip-flop
   END_IF;
   IF #I_AlarmResetPB THEN #SafetySwitchAlm := FALSE; END_IF;
   IF #I_EnableFCAlarm AND #DataFromFC.STW.Warning THEN
       #WarningAlm := TRUE;   // SR flip-flop
   END_IF;
   IF #I_AlarmResetPB THEN #WarningAlm := FALSE; END_IF;
   IF #I_EnableFCAlarm AND #DataFromFC.STW.VoltageLimitExceed THEN
       #VoltageLimitExceedAlm := TRUE;   // SR flip-flop
   END_IF;
   IF #I_AlarmResetPB THEN #VoltageLimitExceedAlm := FALSE; END_IF;
   IF #I_EnableFCAlarm AND #DataFromFC.STW.TorqueLimitExceed THEN
       #TorqueLimitExceedAlm := TRUE;   // SR flip-flop
   END_IF;
   IF #I_AlarmResetPB THEN #TorqueLimitExceedAlm := FALSE; END_IF;
   IF #I_EnableFCAlarm AND #DataFromFC.STW.TimerLimitExceed THEN
       #TimerLimitExceedAlm := TRUE;   // SR flip-flop
   END_IF;
   IF #I_AlarmResetPB THEN #TimerLimitExceedAlm := FALSE; END_IF;
   IF #I_EnableFCAlarm AND #DataFromFC.STW.FrequencyLimit THEN
       #FrequencyLimitAlm := TRUE;   // SR flip-flop
   END_IF;
   IF #I_AlarmResetPB THEN #FrequencyLimitAlm := FALSE; END_IF;
   IF #I_EnableFCAlarm AND (#DataFromFC.PCDIndex3Value > 70) THEN
       #HeatsinkTempAlm := TRUE;   // SR flip-flop
   END_IF;
   IF #I_AlarmResetPB THEN #HeatsinkTempAlm := FALSE; END_IF;
END_REGION

REGION Network 9: **** 5.2 - Equations - Flow Equations **** Frequency controller Active
   // Frequency controller Active
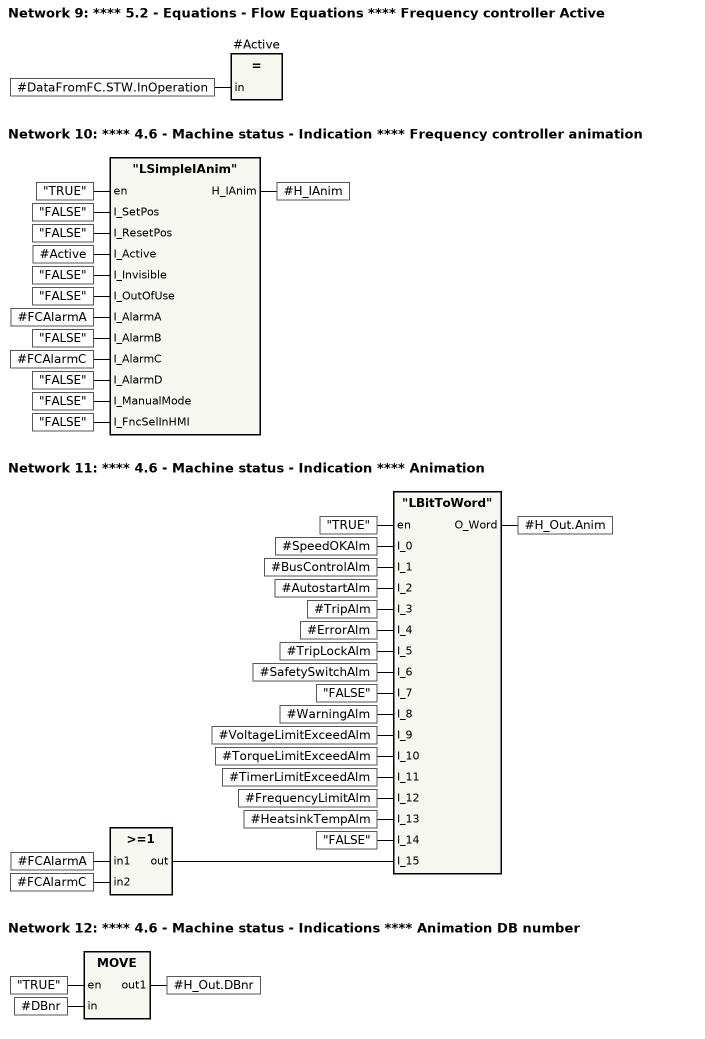
   #Active := #DataFromFC.STW.InOperation;
END_REGION

REGION Network 10: **** 4.6 - Machine status - Indication **** Frequency controller animation
   // Frequency controller animation
   IF "TRUE" THEN
       "LSimpleIAnim"(I_SetPos := "FALSE",
                      I_ResetPos := "FALSE",
                      I_Active := #Active,
                      I_Invisible := "FALSE",
                      I_OutOfUse := "FALSE",
                      I_AlarmA := #FCAlarmA,
                      I_AlarmB := "FALSE",
                      I_AlarmC := #FCAlarmC,
                      I_AlarmD := "FALSE",
                      I_ManualMode := "FALSE",
                      I_FncSelInHMI := "FALSE",
                      H_IAnim => #H_IAnim);
   END_IF;
END_REGION

REGION Network 11: **** 4.6 - Machine status - Indication **** Animation
   // Animation
   IF "TRUE" THEN
       "LBitToWord"(I_0 := #SpeedOKAlm,
                    I_1 := #BusControlAlm,
                    I_2 := #AutostartAlm,
                    I_3 := #TripAlm,
                    I_4 := #ErrorAlm,
                    I_5 := #TripLockAlm,
                    I_6 := #SafetySwitchAlm,
                    I_7 := "FALSE",
                    I_8 := #WarningAlm,
                    I_9 := #VoltageLimitExceedAlm,
                    I_10 := #TorqueLimitExceedAlm,
                    I_11 := #TimerLimitExceedAlm,
                    I_12 := #FrequencyLimitAlm,
                    I_13 := #HeatsinkTempAlm,
                    I_14 := "FALSE",
                    I_15 := #FCAlarmA OR #FCAlarmC,
                    O_Word => #H_Out.Anim);
   END_IF;
END_REGION

REGION Network 12: **** 4.6 - Machine status - Indications **** Animation DB number
   // Animation DB number
   IF "TRUE" THEN #H_Out.DBnr := #DBnr; END_IF;
END_REGION

REGION Network 13: **** 8 - Outputs **** Frequency controller : STW (Status word)
   // Frequency controller : STW (Status word)
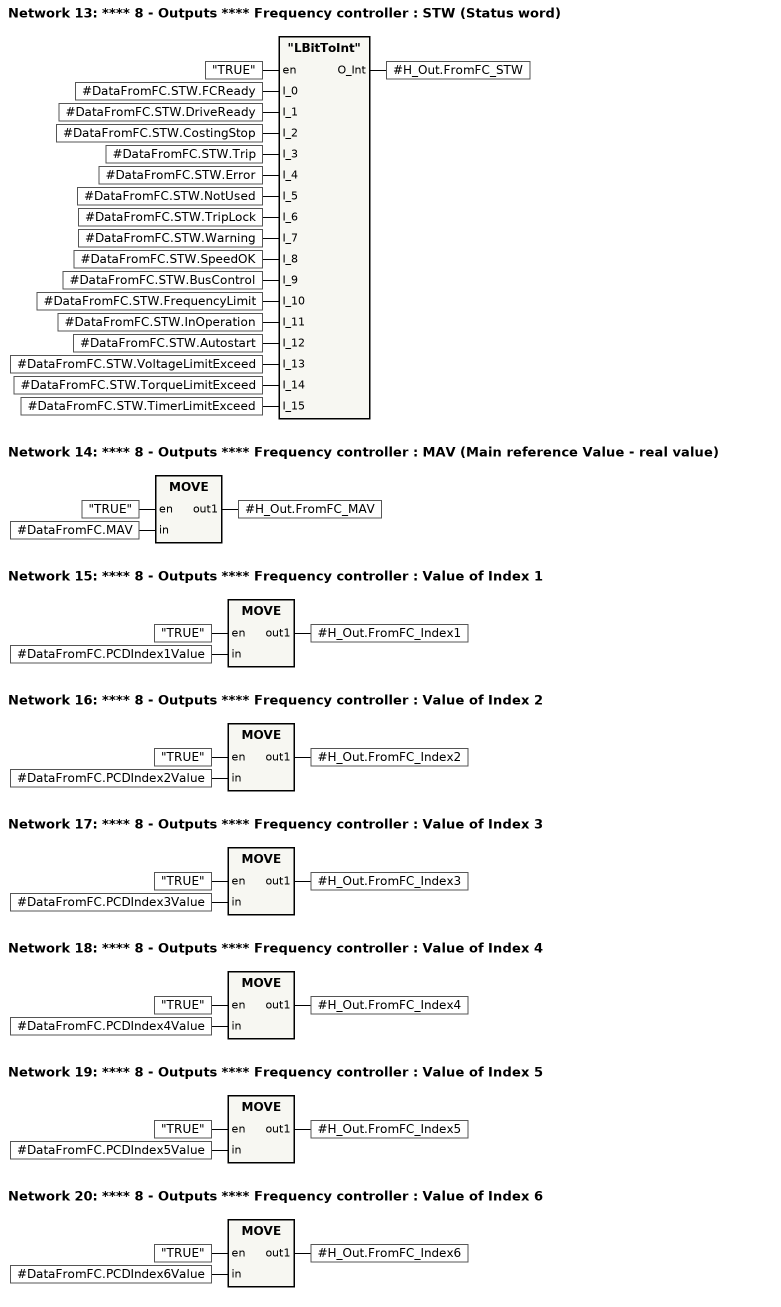
   IF "TRUE" THEN
       "LBitToInt"(I_0 := #DataFromFC.STW.FCReady,
                   I_1 := #DataFromFC.STW.DriveReady,
                   I_2 := #DataFromFC.STW.CostingStop,
                   I_3 := #DataFromFC.STW.Trip,
                   I_4 := #DataFromFC.STW.Error,
                   I_5 := #DataFromFC.STW.NotUsed,
                   I_6 := #DataFromFC.STW.TripLock,
                   I_7 := #DataFromFC.STW.Warning,
                   I_8 := #DataFromFC.STW.SpeedOK,
                   I_9 := #DataFromFC.STW.BusControl,
                   I_10 := #DataFromFC.STW.FrequencyLimit,
                   I_11 := #DataFromFC.STW.InOperation,
                   I_12 := #DataFromFC.STW.Autostart,
                   I_13 := #DataFromFC.STW.VoltageLimitExceed,
                   I_14 := #DataFromFC.STW.TorqueLimitExceed,
                   I_15 := #DataFromFC.STW.TimerLimitExceed,
                   O_Int => #H_Out.FromFC_STW);
   END_IF;
END_REGION

REGION Network 14: **** 8 - Outputs **** Frequency controller : MAV (Main reference Value - real value)
   // Frequency controller : MAV (Main reference Value - real value)
   IF "TRUE" THEN #H_Out.FromFC_MAV := #DataFromFC.MAV; END_IF;
END_REGION

REGION Network 15: **** 8 - Outputs **** Frequency controller : Value of Index 1
   // Frequency controller : Value of Index 1
   IF "TRUE" THEN #H_Out.FromFC_Index1 := #DataFromFC.PCDIndex1Value; END_IF;
END_REGION

REGION Network 16: **** 8 - Outputs **** Frequency controller : Value of Index 2
   // Frequency controller : Value of Index 2
   IF "TRUE" THEN #H_Out.FromFC_Index2 := #DataFromFC.PCDIndex2Value; END_IF;
END_REGION

REGION Network 17: **** 8 - Outputs **** Frequency controller : Value of Index 3
   // Frequency controller : Value of Index 3
   IF "TRUE" THEN #H_Out.FromFC_Index3 := #DataFromFC.PCDIndex3Value; END_IF;
END_REGION

REGION Network 18: **** 8 - Outputs **** Frequency controller : Value of Index 4
   // Frequency controller : Value of Index 4
   IF "TRUE" THEN #H_Out.FromFC_Index4 := #DataFromFC.PCDIndex4Value; END_IF;
END_REGION

REGION Network 19: **** 8 - Outputs **** Frequency controller : Value of Index 5
   // Frequency controller : Value of Index 5
   IF "TRUE" THEN #H_Out.FromFC_Index5 := #DataFromFC.PCDIndex5Value; END_IF;
END_REGION

REGION Network 20: **** 8 - Outputs **** Frequency controller : Value of Index 6
   // Frequency controller : Value of Index 6
   IF "TRUE" THEN #H_Out.FromFC_Index6 := #DataFromFC.PCDIndex6Value; END_IF;
END_REGION

REGION Network 21: **** 8 - Outputs **** Frequency controller : Value of Index 7
   // Frequency controller : Value of Index 7
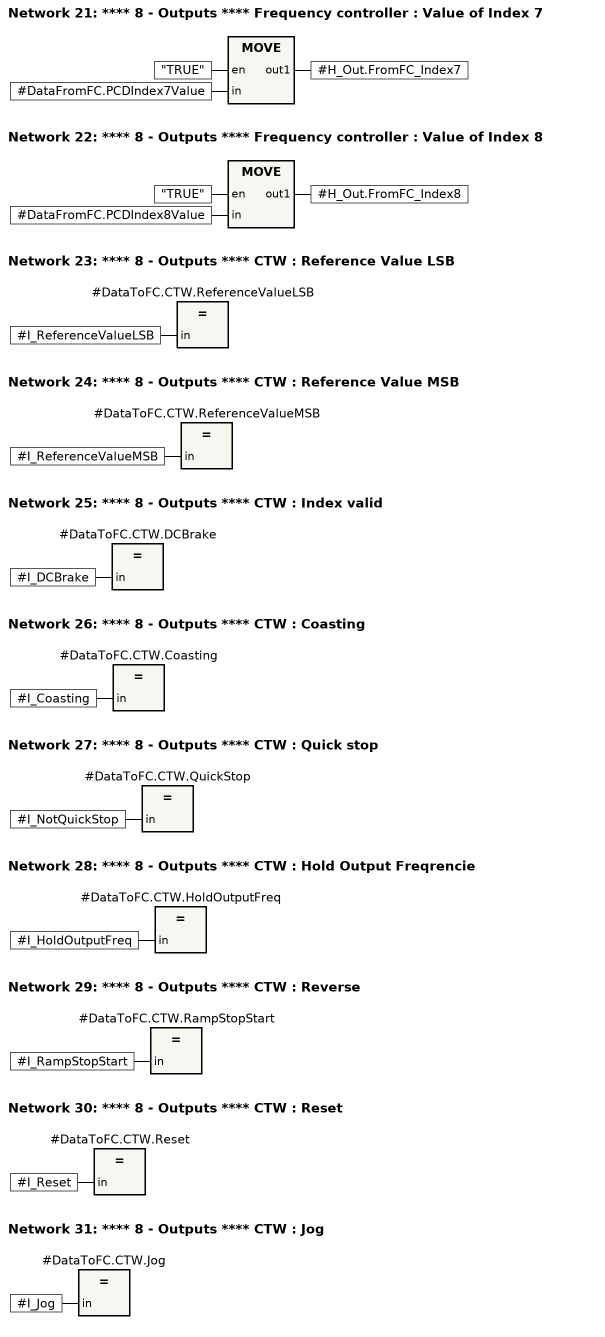
   IF "TRUE" THEN #H_Out.FromFC_Index7 := #DataFromFC.PCDIndex7Value; END_IF;
END_REGION

REGION Network 22: **** 8 - Outputs **** Frequency controller : Value of Index 8
   // Frequency controller : Value of Index 8
   IF "TRUE" THEN #H_Out.FromFC_Index8 := #DataFromFC.PCDIndex8Value; END_IF;
END_REGION

REGION Network 23: **** 8 - Outputs **** CTW : Reference Value LSB
   // CTW : Reference Value LSB
   #DataToFC.CTW.ReferenceValueLSB := #I_ReferenceValueLSB;
END_REGION

REGION Network 24: **** 8 - Outputs **** CTW : Reference Value MSB
   // CTW : Reference Value MSB
   #DataToFC.CTW.ReferenceValueMSB := #I_ReferenceValueMSB;
END_REGION

REGION Network 25: **** 8 - Outputs **** CTW : Index valid
   // CTW : Index valid
   #DataToFC.CTW.DCBrake := #I_DCBrake;
END_REGION

REGION Network 26: **** 8 - Outputs **** CTW : Coasting
   // CTW : Coasting
   #DataToFC.CTW.Coasting := #I_Coasting;
END_REGION

REGION Network 27: **** 8 - Outputs **** CTW : Quick stop
   // CTW : Quick stop
   #DataToFC.CTW.QuickStop := #I_NotQuickStop;
END_REGION

REGION Network 28: **** 8 - Outputs **** CTW : Hold Output Freqrencie
   // CTW : Hold Output Freqrencie
   #DataToFC.CTW.HoldOutputFreq := #I_HoldOutputFreq;
END_REGION

REGION Network 29: **** 8 - Outputs **** CTW : Reverse
   // CTW : Reverse
   #DataToFC.CTW.RampStopStart := #I_RampStopStart;
END_REGION

REGION Network 30: **** 8 - Outputs **** CTW : Reset
   // CTW : Reset
   #DataToFC.CTW.Reset := #I_Reset;
END_REGION

REGION Network 31: **** 8 - Outputs **** CTW : Jog
   // CTW : Jog
   #DataToFC.CTW.Jog := #I_Jog;
END_REGION

REGION Network 32: **** 8 - Outputs **** CTW : Ramp Selection
   // CTW : Ramp Selection
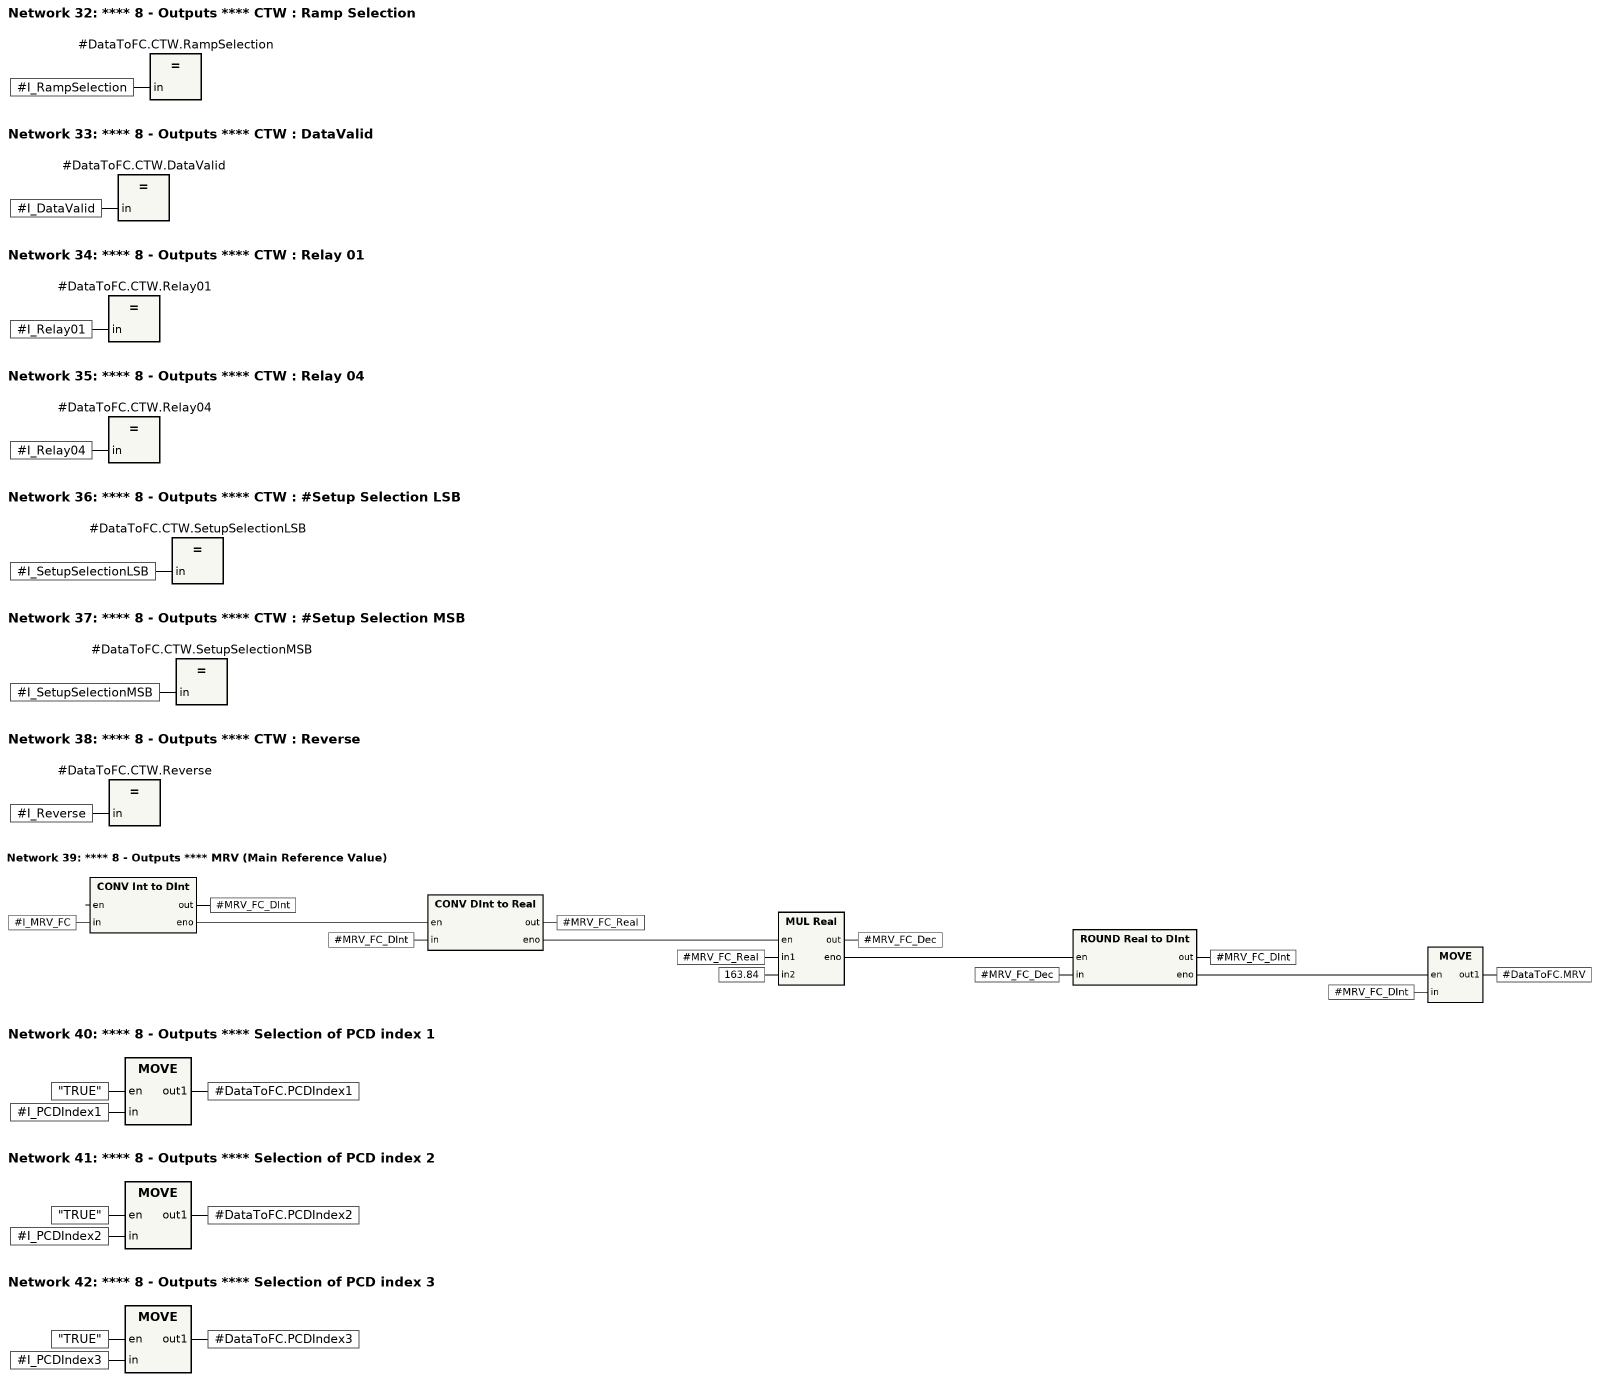
   #DataToFC.CTW.RampSelection := #I_RampSelection;
END_REGION

REGION Network 33: **** 8 - Outputs **** CTW : DataValid
   // CTW : DataValid
   #DataToFC.CTW.DataValid := #I_DataValid;
END_REGION

REGION Network 34: **** 8 - Outputs **** CTW : Relay 01
   // CTW : Relay 01
   #DataToFC.CTW.Relay01 := #I_Relay01;
END_REGION

REGION Network 35: **** 8 - Outputs **** CTW : Relay 04
   // CTW : Relay 04
   #DataToFC.CTW.Relay04 := #I_Relay04;
END_REGION

REGION Network 36: **** 8 - Outputs **** CTW : #Setup Selection LSB
   // CTW : #Setup Selection LSB
   #DataToFC.CTW.SetupSelectionLSB := #I_SetupSelectionLSB;
END_REGION

REGION Network 37: **** 8 - Outputs **** CTW : #Setup Selection MSB
   // CTW : #Setup Selection MSB
   #DataToFC.CTW.SetupSelectionMSB := #I_SetupSelectionMSB;
END_REGION

REGION Network 38: **** 8 - Outputs **** CTW : Reverse
   // CTW : Reverse
   #DataToFC.CTW.Reverse := #I_Reverse;
END_REGION

REGION Network 39: **** 8 - Outputs **** MRV (Main Reference Value)
   // MRV (Main Reference Value)
   // ENO of a box is taken as its EN; it also drops when the box reports an error
   #MRV_FC_DInt := INT_TO_DINT(#I_MRV_FC);
   #MRV_FC_Real := DINT_TO_REAL(#MRV_FC_DInt);
   #MRV_FC_Dec := #MRV_FC_Real * 163.84;
   #MRV_FC_DInt := ROUND(#MRV_FC_Dec);
   #DataToFC.MRV := #MRV_FC_DInt;
END_REGION

REGION Network 40: **** 8 - Outputs **** Selection of PCD index 1
   // Selection of PCD index 1
   IF "TRUE" THEN #DataToFC.PCDIndex1 := #I_PCDIndex1; END_IF;
END_REGION

REGION Network 41: **** 8 - Outputs **** Selection of PCD index 2
   // Selection of PCD index 2
   IF "TRUE" THEN #DataToFC.PCDIndex2 := #I_PCDIndex2; END_IF;
END_REGION

REGION Network 42: **** 8 - Outputs **** Selection of PCD index 3
   // Selection of PCD index 3
   IF "TRUE" THEN #DataToFC.PCDIndex3 := #I_PCDIndex3; END_IF;
END_REGION

REGION Network 43: **** 8 - Outputs **** Selection of PCD index 4
   // Selection of PCD index 4
